LIN {X 0,Y 225.731,Z 1154.757,A -85,B 0,C 180,E1 26958.858,E2 26958.858} C_VEL
LIN {X 0,Y 255.591,Z 1130.454,A -85,B 0,C 180,E1 26969.522,E2 26969.522} C_VEL
LIN {X 0,Y 287.128,Z 1102.716,A -85,B 0,C 180,E1 26976.829,E2 26976.829} C_VEL
LIN {X 0,Y 319.743,Z 1070.349,A -85,B 0,C 180,E1 26982.239,E2 26982.239} C_VEL
LIN {X 0,Y 351.909,Z 1032.611,A -85,B 0,C 180,E1 26986.269,E2 26986.269} C_VEL
LIN {X 0,Y 368.371,Z 1010.613,A -85,B 0,C 180,E1 26987.946,E2 26987.946} C_VEL
LIN {X 0,Y 369.064,Z 1007.37,A -85,B 0,C 180,E1 26989.314,E2 26989.314} C_VEL
LIN {X 0,Y 369.295,Z 1000.148,A -85,B 0,C 180,E1 26995.312,E2 26995.312} C_VEL
LIN {X 0,Y 369.425,Z 998.78,A -85,B 0,C 180,E1 26997.662,E2 26997.662} C_VEL
LIN {X 0,Y 368.67,Z 999.428,A -85,B 0,C 180,E1 27000.006,E2 27000.006} C_VEL
LIN {X 0,Y 365.941,Z 1005.713,A -85,B 0,C 180,E1 27005.933,E2 27005.933} C_VEL
LIN {X 0,Y 364.301,Z 1009.952,A -85,B 0,C 180,E1 27008.244,E2 27008.244} C_VEL
LIN {X 0,Y 336.486,Z 1043.678,A -85,B 0,C 180,E1 27011.534,E2 27011.534} C_VEL
LIN {X 0,Y 304.444,Z 1075.769,A -85,B 0,C 180,E1 27016.292,E2 27016.292} C_VEL
LIN {X 0,Y 273.32,Z 1102.243,A -85,B 0,C 180,E1 27022.45,E2 27022.45} C_VEL
LIN {X 0,Y 242.415,Z 1124.929,A -85,B 0,C 180,E1 27031.225,E2 27031.225} C_VEL
LIN {X 0,Y 228.244,Z 1134.299,A -85,B 0,C 180,E1 27036.811,E2 27036.811} C_VEL
LIN {X 0,Y 217.232,Z 1139.855,A -85,B 0,C 180,E1 27040.027,E2 27040.027} C_VEL
LIN {X 0,Y 206.835,Z 1144.678,A -85,B 0,C 180,E1 27043.615,E2 27043.615} C_VEL
LIN {X 0,Y 192.084,Z 1153.208,A -85,B 0,C 180,E1 27056.588,E2 27056.588} C_VEL
LIN {X 0,Y 184.823,Z 1157.192,A -85,B 0,C 180,E1 27070.913,E2 27070.913} C_VEL
LIN {X 0,Y 183.688,Z 1157.067,A -85,B 0,C 180,E1 27080.911,E2 27080.911} C_VEL
LIN {X 0,Y 184.934,Z 1155.178,A -85,B 0,C 180,E1 27090.002,E2 27090.002} C_VEL
LIN {X 0,Y 189.195,Z 1150.026,A -85,B 0,C 180,E1 27101.521,E2 27101.521} C_VEL
LIN {X 0,Y 199.74,Z 1139.824,A -85,B 0,C 180,E1 27114.27,E2 27114.27} C_VEL
LIN {X 0,Y 218.512,Z 1123.996,A -85,B 0,C 180,E1 27126.005,E2 27126.005} C_VEL
LIN {X 0,Y 244.526,Z 1101.275,A -85,B 0,C 180,E1 27135.925,E2 27135.925} C_VEL
LIN {X 0,Y 271.832,Z 1074.958,A -85,B 0,C 180,E1 27143.048,E2 27143.048} C_VEL
LIN {X 0,Y 300.799,Z 1042.826,A -85,B 0,C 180,E1 27148.655,E2 27148.655} C_VEL
LIN {X 0,Y 327.326,Z 1007.742,A -85,B 0,C 180,E1 27152.712,E2 27152.712} C_VEL
LIN {X 0,Y 337.468,Z 992.575,A -85,B 0,C 180,E1 27154.024,E2 27154.024} C_VEL
LIN {X 0,Y 339.323,Z 979.812,A -85,B 0,C 180,E1 27159.121,E2 27159.121} C_VEL
LIN {X 0,Y 340.418,Z 970.596,A -85,B 0,C 180,E1 27164.546,E2 27164.546} C_VEL
LIN {X 0,Y 341.292,Z 965.531,A -85,B 0,C 180,E1 27169.791,E2 27169.791} C_VEL
LIN {X 0,Y 342.341,Z 964.643,A -85,B 0,C 180,E1 27174.928,E2 27174.928} C_VEL
LIN {X 0,Y 342.913,Z 967.181,A -85,B 0,C 180,E1 27178.73,E2 27178.73} C_VEL
LIN {X 0,Y 343.424,Z 975.954,A -85,B 0,C 180,E1 27184.409,E2 27184.409} C_VEL
LIN {X 0,Y 343.453,Z 988.167,A -85,B 0,C 180,E1 27189.49,E2 27189.49} C_VEL
LIN {X 0,Y 342.79,Z 996.133,A -85,B 0,C 180,E1 27191.913,E2 27191.913} C_VEL
LIN {X 0,Y 317.01,Z 1035.287,A -85,B 0,C 180,E1 27195.203,E2 27195.203} C_VEL
LIN {X 0,Y 288.961,Z 1071.469,A -85,B 0,C 180,E1 27199.722,E2 27199.722} C_VEL
LIN {X 0,Y 259.817,Z 1103.901,A -85,B 0,C 180,E1 27205.948,E2 27205.948} C_VEL
LIN {X 0,Y 232.582,Z 1131.307,A -85,B 0,C 180,E1 27214.063,E2 27214.063} C_VEL
LIN {X 0,Y 208.777,Z 1154.112,A -85,B 0,C 180,E1 27224.97,E2 27224.97} C_VEL
LIN {X 0,Y 193.756,Z 1169.833,A -85,B 0,C 180,E1 27236.909,E2 27236.909} C_VEL
LIN {X 0,Y 186.533,Z 1179.298,A -85,B 0,C 180,E1 27248.16,E2 27248.16} C_VEL
LIN {X 0,Y 183.801,Z 1185.477,A -85,B 0,C 180,E1 27260.533,E2 27260.533} C_VEL
LIN {X 0,Y 184.143,Z 1187.355,A -85,B 0,C 180,E1 27269.998,E2 27269.998} C_VEL
LIN {X 0,Y 183.626,Z 1186.803,A -85,B 0,C 180,E1 27279.471,E2 27279.471} C_VEL
LIN {X 0,Y 187.317,Z 1181.478,A -85,B 0,C 180,E1 27293.786,E2 27293.786} C_VEL
LIN {X 0,Y 199.841,Z 1170.086,A -85,B 0,C 180,E1 27308.594,E2 27308.594} C_VEL
LIN {X 0,Y 220.297,Z 1154.314,A -85,B 0,C 180,E1 27320.475,E2 27320.475} C_VEL
LIN {X 0,Y 250.559,Z 1130.739,A -85,B 0,C 180,E1 27330.922,E2 27330.922} C_VEL
LIN {X 0,Y 282.961,Z 1103.312,A -85,B 0,C 180,E1 27338.19,E2 27338.19} C_VEL
LIN {X 0,Y 316.996,Z 1070.447,A -85,B 0,C 180,E1 27343.605,E2 27343.605} C_VEL
LIN {X 0,Y 348.412,Z 1034.569,A -85,B 0,C 180,E1 27347.387,E2 27347.387} C_VEL
LIN {X 0,Y 363.267,Z 1015.279,A -85,B 0,C 180,E1 27348.857,E2 27348.857} C_VEL
LIN {X 0,Y 364.088,Z 1012.889,A -85,B 0,C 180,E1 27349.809,E2 27349.809} C_VEL
LIN {X 0,Y 364.525,Z 1006.563,A -85,B 0,C 180,E1 27355.251,E2 27355.251} C_VEL
LIN {X 0,Y 364.682,Z 1005.142,A -85,B 0,C 180,E1 27357.632,E2 27357.632} C_VEL
LIN {X 0,Y 362.859,Z 1007.313,A -85,B 0,C 180,E1 27361.884,E2 27361.884} C_VEL
LIN {X 0,Y 360.058,Z 1014.019,A -85,B 0,C 180,E1 27367.24,E2 27367.24} C_VEL
LIN {X 0,Y 330.698,Z 1048.189,A -85,B 0,C 180,E1 27370.659,E2 27370.659} C_VEL
LIN {X 0,Y 297.895,Z 1079.882,A -85,B 0,C 180,E1 27375.467,E2 27375.467} C_VEL
LIN {X 0,Y 266.374,Z 1105.375,A -85,B 0,C 180,E1 27381.653,E2 27381.653} C_VEL
LIN {X 0,Y 236.474,Z 1126.44,A -85,B 0,C 180,E1 27390.032,E2 27390.032} C_VEL
LIN {X 0,Y 210.577,Z 1142.41,A -85,B 0,C 180,E1 27401.326,E2 27401.326} C_VEL
LIN {X 0,Y 206.835,Z 1144.678,A -85,B 0,C 180,E1 27403.615,E2 27403.615} C_VEL
LIN {X 0,Y 197.08,Z 1148.854,A -85,B 0,C 180,E1 27407.583,E2 27407.583} C_VEL
LIN {X 0,Y 188.062,Z 1152.273,A -85,B 0,C 180,E1 27411.94,E2 27411.94} C_VEL
LIN {X 0,Y 178.94,Z 1157.001,A -85,B 0,C 180,E1 27425.026,E2 27425.026} C_VEL
LIN {X 0,Y 176.095,Z 1158.029,A -85,B 0,C 180,E1 27435.084,E2 27435.084} C_VEL
LIN {X 0,Y 176.124,Z 1157.066,A -85,B 0,C 180,E1 27445.08,E2 27445.08} C_VEL
LIN {X 0,Y 179.237,Z 1153.177,A -85,B 0,C 180,E1 27457.268,E2 27457.268} C_VEL
LIN {X 0,Y 188.287,Z 1144.419,A -85,B 0,C 180,E1 27471.174,E2 27471.174} C_VEL
LIN {X 0,Y 205.027,Z 1130.704,A -85,B 0,C 180,E1 27483.56,E2 27483.56} C_VEL
LIN {X 0,Y 231.034,Z 1109.426,A -85,B 0,C 180,E1 27494.681,E2 27494.681} C_VEL
LIN {X 0,Y 259.187,Z 1083.962,A -85,B 0,C 180,E1 27502.599,E2 27502.599} C_VEL
LIN {X 0,Y 287.826,Z 1054.539,A -85,B 0,C 180,E1 27508.413,E2 27508.413} C_VEL
LIN {X 0,Y 317.766,Z 1017.751,A -85,B 0,C 180,E1 27513.119,E2 27513.119} C_VEL
LIN {X 0,Y 332.912,Z 995.879,A -85,B 0,C 180,E1 27515.209,E2 27515.209} C_VEL
LIN {X 0,Y 334.922,Z 984.233,A -85,B 0,C 180,E1 27520.277,E2 27520.277} C_VEL
LIN {X 0,Y 336.156,Z 975.928,A -85,B 0,C 180,E1 27525.678,E2 27525.678} C_VEL
LIN {X 0,Y 337.207,Z 972.067,A -85,B 0,C 180,E1 27530.37,E2 27530.37} C_VEL
LIN {X 0,Y 338.186,Z 971.363,A -85,B 0,C 180,E1 27534.866,E2 27534.866} C_VEL
LIN {X 0,Y 338.706,Z 973.965,A -85,B 0,C 180,E1 27538.715,E2 27538.715} C_VEL
LIN {X 0,Y 338.891,Z 982.852,A -85,B 0,C 180,E1 27544.469,E2 27544.469} C_VEL
LIN {X 0,Y 338.543,Z 995.446,A -85,B 0,C 180,E1 27549.629,E2 27549.629} C_VEL
LIN {X 0,Y 337.882,Z 999.689,A -85,B 0,C 180,E1 27550.903,E2 27550.903} C_VEL
LIN {X 0,Y 309.246,Z 1041.451,A -85,B 0,C 180,E1 27554.497,E2 27554.497} C_VEL
LIN {X 0,Y 279.64,Z 1077.497,A -85,B 0,C 180,E1 27559.272,E2 27559.272} C_VEL
LIN {X 0,Y 251.113,Z 1107.96,A -85,B 0,C 180,E1 27565.486,E2 27565.486} C_VEL
LIN {X 0,Y 222.993,Z 1134.715,A -85,B 0,C 180,E1 27574.064,E2 27574.064} C_VEL
LIN {X 0,Y 199.803,Z 1156.182,A -85,B 0,C 180,E1 27585.154,E2 27585.154} C_VEL
LIN {X 0,Y 183.614,Z 1172.48,A -85,B 0,C 180,E1 27599.322,E2 27599.322} C_VEL
LIN {X 0,Y 177.133,Z 1181.607,A -85,B 0,C 180,E1 27612.625,E2 27612.625} C_VEL
LIN {X 0,Y 175.787,Z 1185.998,A -85,B 0,C 180,E1 27625.066,E2 27625.066} C_VEL
LIN {X 0,Y 176.27,Z 1186.693,A -85,B 0,C 180,E1 27629.998,E2 27629.998} C_VEL
LIN {X 0,Y 175.744,Z 1186.154,A -85,B 0,C 180,E1 27639.9,E2 27639.9} C_VEL
LIN {X 0,Y 179.846,Z 1180.886,A -85,B 0,C 180,E1 27654.839,E2 27654.839} C_VEL
LIN {X 0,Y 193.381,Z 1169.535,A -85,B 0,C 180,E1 27670.138,E2 27670.138} C_VEL
LIN {X 0,Y 216.929,Z 1152.407,A -85,B 0,C 180,E1 27683,E2 27683} C_VEL
LIN {X 0,Y 247.722,Z 1129.486,A -85,B 0,C 180,E1 27692.909,E2 27692.909} C_VEL
LIN {X 0,Y 280.898,Z 1102.184,A -85,B 0,C 180,E1 27699.931,E2 27699.931} C_VEL
LIN {X 0,Y 314.777,Z 1070.205,A -85,B 0,C 180,E1 27705.039,E2 27705.039} C_VEL
LIN {X 0,Y 346.723,Z 1034.468,A -85,B 0,C 180,E1 27708.702,E2 27708.702} C_VEL
LIN {X 0,Y 358.957,Z 1018.778,A -85,B 0,C 180,E1 27710.007,E2 27710.007} C_VEL
LIN {X 0,Y 359.519,Z 1012.804,A -85,B 0,C 180,E1 27715.184,E2 27715.184} C_VEL
LIN {X 0,Y 359.717,Z 1011.351,A -85,B 0,C 180,E1 27717.599,E2 27717.599} C_VEL
LIN {X 0,Y 358.821,Z 1012.013,A -85,B 0,C 180,E1 27720.007,E2 27720.007} C_VEL
LIN {X 0,Y 355.697,Z 1018.071,A -85,B 0,C 180,E1 27725.824,E2 27725.824} C_VEL
LIN {X 0,Y 354.503,Z 1019.844,A -85,B 0,C 180,E1 27726.44,E2 27726.44} C_VEL
LIN {X 0,Y 324.04,Z 1053.622,A -85,B 0,C 180,E1 27729.87,E2 27729.87} C_VEL
LIN {X 0,Y 293.44,Z 1082.113,A -85,B 0,C 180,E1 27734.272,E2 27734.272} C_VEL
LIN {X 0,Y 258.884,Z 1108.955,A -85,B 0,C 180,E1 27740.948,E2 27740.948} C_VEL
LIN {X 0,Y 228.53,Z 1129.114,A -85,B 0,C 180,E1 27749.483,E2 27749.483} C_VEL
LIN {X 0,Y 201.7,Z 1144.875,A -85,B 0,C 180,E1 27761.482,E2 27761.482} C_VEL
LIN {X 0,Y 188.062,Z 1152.273,A -85,B 0,C 180,E1 27771.94,E2 27771.94} C_VEL
LIN {X 0,Y 182.293,Z 1154.397,A -85,B 0,C 180,E1 27775.515,E2 27775.515} C_VEL
LIN {X 0,Y 173.01,Z 1156.924,A -85,B 0,C 180,E1 27781.105,E2 27781.105} C_VEL
LIN {X 0,Y 172.518,Z 1157.109,A -85,B 0,C 180,E1 27781.812,E2 27781.812} C_VEL
LIN {X 0,Y 168.284,Z 1158.679,A -85,B 0,C 180,E1 27794.375,E2 27794.375} C_VEL
LIN {X 0,Y 168.189,Z 1157.771,A -85,B 0,C 180,E1 27804.848,E2 27804.848} C_VEL
LIN {X 0,Y 171.444,Z 1153.939,A -85,B 0,C 180,E1 27817.6,E2 27817.6} C_VEL
LIN {X 0,Y 180.976,Z 1145.25,A -85,B 0,C 180,E1 27832.073,E2 27832.073} C_VEL
LIN {X 0,Y 198.518,Z 1131.649,A -85,B 0,C 180,E1 27844.816,E2 27844.816} C_VEL
LIN {X 0,Y 225.53,Z 1110.45,A -85,B 0,C 180,E1 27856.081,E2 27856.081} C_VEL
LIN {X 0,Y 254.512,Z 1085.139,A -85,B 0,C 180,E1 27863.998,E2 27863.998} C_VEL
LIN {X 0,Y 284.131,Z 1055.549,A -85,B 0,C 180,E1 27869.799,E2 27869.799} C_VEL
LIN {X 0,Y 314.371,Z 1019.202,A -85,B 0,C 180,E1 27874.382,E2 27874.382} C_VEL
LIN {X 0,Y 327.409,Z 1001.32,A -85,B 0,C 180,E1 27876.004,E2 27876.004} C_VEL
LIN {X 0,Y 328.56,Z 998.218,A -85,B 0,C 180,E1 27876.907,E2 27876.907} C_VEL
LIN {X 0,Y 330.956,Z 986.563,A -85,B 0,C 180,E1 27882.729,E2 27882.729} C_VEL
LIN {X 0,Y 332.263,Z 980.103,A -85,B 0,C 180,E1 27888.183,E2 27888.183} C_VEL
LIN {X 0,Y 333.478,Z 978.043,A -85,B 0,C 180,E1 27893.438,E2 27893.438} C_VEL
LIN {X 0,Y 334.375,Z 979.22,A -85,B 0,C 180,E1 27897.403,E2 27897.403} C_VEL
LIN {X 0,Y 334.251,Z 987.229,A -85,B 0,C 180,E1 27903.233,E2 27903.233} C_VEL
LIN {X 0,Y 333.666,Z 998.99,A -85,B 0,C 180,E1 27908.457,E2 27908.457} C_VEL
LIN {X 0,Y 333.359,Z 1002.551,A -85,B 0,C 180,E1 27909.78,E2 27909.78} C_VEL
LIN {X 0,Y 304.76,Z 1043.252,A -85,B 0,C 180,E1 27913.316,E2 27913.316} C_VEL
LIN {X 0,Y 273.281,Z 1080.243,A -85,B 0,C 180,E1 27918.274,E2 27918.274} C_VEL
LIN {X 0,Y 243.35,Z 1110.799,A -85,B 0,C 180,E1 27924.742,E2 27924.742} C_VEL
LIN {X 0,Y 213.562,Z 1137.974,A -85,B 0,C 180,E1 27934.001,E2 27934.001} C_VEL
LIN {X 0,Y 190.625,Z 1158.131,A -85,B 0,C 180,E1 27945.5,E2 27945.5} C_VEL
LIN {X 0,Y 175.419,Z 1172.928,A -85,B 0,C 180,E1 27959.454,E2 27959.454} C_VEL
LIN {X 0,Y 169.44,Z 1180.852,A -85,B 0,C 180,E1 27971.809,E2 27971.809} C_VEL
LIN {X 0,Y 167.885,Z 1185.307,A -85,B 0,C 180,E1 27984.833,E2 27984.833} C_VEL
LIN {X 0,Y 168.375,Z 1186.03,A -85,B 0,C 180,E1 27989.997,E2 27989.997} C_VEL
LIN {X 0,Y 167.888,Z 1185.507,A -85,B 0,C 180,E1 28000.368,E2 28000.368} C_VEL
LIN {X 0,Y 172.441,Z 1180.296,A -85,B 0,C 180,E1 28015.984,E2 28015.984} C_VEL
LIN {X 0,Y 187.013,Z 1169.049,A -85,B 0,C 180,E1 28031.715,E2 28031.715} C_VEL
LIN {X 0,Y 210.887,Z 1152.735,A -85,B 0,C 180,E1 28044.367,E2 28044.367} C_VEL
LIN {X 0,Y 244.692,Z 1128.602,A -85,B 0,C 180,E1 28054.817,E2 28054.817} C_VEL
LIN {X 0,Y 278.629,Z 1101.448,A -85,B 0,C 180,E1 28061.631,E2 28061.631} C_VEL
LIN {X 0,Y 314.428,Z 1068.351,A -85,B 0,C 180,E1 28066.701,E2 28066.701} C_VEL
LIN {X 0,Y 348.48,Z 1030.407,A -85,B 0,C 180,E1 28070.341,E2 28070.341} C_VEL
LIN {X 0,Y 353.938,Z 1023.696,A -85,B 0,C 180,E1 28070.868,E2 28070.868} C_VEL
LIN {X 0,Y 354.461,Z 1019.006,A -85,B 0,C 180,E1 28075.115,E2 28075.115} C_VEL
LIN {X 0,Y 354.688,Z 1017.501,A -85,B 0,C 180,E1 28077.565,E2 28077.565} C_VEL
LIN {X 0,Y 353.016,Z 1019.198,A -85,B 0,C 180,E1 28081.233,E2 28081.233} C_VEL
LIN {X 0,Y 350.663,Z 1023.307,A -85,B 0,C 180,E1 28085.231,E2 28085.231} C_VEL
LIN {X 0,Y 319.094,Z 1057.396,A -85,B 0,C 180,E1 28088.854,E2 28088.854} C_VEL
LIN {X 0,Y 285.521,Z 1087.118,A -85,B 0,C 180,E1 28093.605,E2 28093.605} C_VEL
LIN {X 0,Y 253.013,Z 1111.397,A -85,B 0,C 180,E1 28099.843,E2 28099.843} C_VEL
LIN {X 0,Y 221.711,Z 1131.129,A -85,B 0,C 180,E1 28108.509,E2 28108.509} C_VEL
LIN {X 0,Y 196.209,Z 1145.373,A -85,B 0,C 180,E1 28119.635,E2 28119.635} C_VEL
LIN {X 0,Y 178.328,Z 1154.355,A -85,B 0,C 180,E1 28133.621,E2 28133.621} C_VEL
LIN {X 0,Y 172.518,Z 1157.109,A -85,B 0,C 180,E1 28141.812,E2 28141.812} C_VEL
LIN {X 0,Y 167.988,Z 1158.233,A -85,B 0,C 180,E1 28145.949,E2 28145.949} C_VEL
LIN {X 0,Y 160.783,Z 1159.292,A -85,B 0,C 180,E1 28152.412,E2 28152.412} C_VEL
LIN {X 0,Y 160.57,Z 1159.316,A -85,B 0,C 180,E1 28153.195,E2 28153.195} C_VEL
LIN {X 0,Y 160.265,Z 1158.474,A -85,B 0,C 180,E1 28164.592,E2 28164.592} C_VEL
LIN {X 0,Y 163.674,Z 1154.698,A -85,B 0,C 180,E1 28177.963,E2 28177.963} C_VEL
LIN {X 0,Y 173.716,Z 1146.077,A -85,B 0,C 180,E1 28193.047,E2 28193.047} C_VEL
LIN {X 0,Y 192.116,Z 1132.592,A -85,B 0,C 180,E1 28206.155,E2 28206.155} C_VEL
LIN {X 0,Y 220.164,Z 1111.474,A -85,B 0,C 180,E1 28217.551,E2 28217.551} C_VEL
LIN {X 0,Y 249.998,Z 1086.315,A -85,B 0,C 180,E1 28225.447,E2 28225.447} C_VEL
LIN {X 0,Y 280.296,Z 1056.832,A -85,B 0,C 180,E1 28231.175,E2 28231.175} C_VEL
LIN {X 0,Y 310.571,Z 1021.366,A -85,B 0,C 180,E1 28235.6,E2 28235.6} C_VEL
LIN {X 0,Y 323.505,Z 1003.782,A -85,B 0,C 180,E1 28237.325,E2 28237.325} C_VEL
LIN {X 0,Y 326.234,Z 992.448,A -85,B 0,C 180,E1 28243.148,E2 28243.148} C_VEL
LIN {X 0,Y 327.846,Z 986.527,A -85,B 0,C 180,E1 28248.396,E2 28248.396} C_VEL
LIN {X 0,Y 329.032,Z 984.615,A -85,B 0,C 180,E1 28253.473,E2 28253.473} C_VEL
LIN {X 0,Y 329.875,Z 985.796,A -85,B 0,C 180,E1 28257.367,E2 28257.367} C_VEL
LIN {X 0,Y 329.614,Z 994.014,A -85,B 0,C 180,E1 28263.278,E2 28263.278} C_VEL
LIN {X 0,Y 328.439,Z 1006.01,A -85,B 0,C 180,E1 28268.593,E2 28268.593} C_VEL
LIN {X 0,Y 322.913,Z 1014.638,A -85,B 0,C 180,E1 28269.365,E2 28269.365} C_VEL
LIN {X 0,Y 293.321,Z 1053.597,A -85,B 0,C 180,E1 28273.105,E2 28273.105} C_VEL
LIN {X 0,Y 263.005,Z 1087.06,A -85,B 0,C 180,E1 28277.975,E2 28277.975} C_VEL
LIN {X 0,Y 230.898,Z 1117.905,A -85,B 0,C 180,E1 28285.168,E2 28285.168} C_VEL
LIN {X 0,Y 202.269,Z 1142.521,A -85,B 0,C 180,E1 28294.731,E2 28294.731} C_VEL
LIN {X 0,Y 179.093,Z 1162.144,A -85,B 0,C 180,E1 28307.542,E2 28307.542} C_VEL
LIN {X 0,Y 165.168,Z 1175.494,A -85,B 0,C 180,E1 28322.774,E2 28322.774} C_VEL
LIN {X 0,Y 161.072,Z 1181.398,A -85,B 0,C 180,E1 28333.65,E2 28333.65} C_VEL
LIN {X 0,Y 160.001,Z 1184.616,A -85,B 0,C 180,E1 28344.578,E2 28344.578} C_VEL
LIN {X 0,Y 160.497,Z 1185.368,A -85,B 0,C 180,E1 28349.997,E2 28349.997} C_VEL
LIN {X 0,Y 160.014,Z 1184.857,A -85,B 0,C 180,E1 28360.884,E2 28360.884} C_VEL
LIN {X 0,Y 163.659,Z 1180.889,A -85,B 0,C 180,E1 28374.548,E2 28374.548} C_VEL
LIN {X 0,Y 177.039,Z 1171.082,A -85,B 0,C 180,E1 28390.629,E2 28390.629} C_VEL
LIN {X 0,Y 202.91,Z 1154.305,A -85,B 0,C 180,E1 28405.001,E2 28405.001} C_VEL
LIN {X 0,Y 233.771,Z 1133.521,A -85,B 0,C 180,E1 28414.816,E2 28414.816} C_VEL
LIN {X 0,Y 271.366,Z 1105.178,A -85,B 0,C 180,E1 28422.476,E2 28422.476} C_VEL
LIN {X 0,Y 306.396,Z 1074.104,A -85,B 0,C 180,E1 28427.433,E2 28427.433} C_VEL
LIN {X 0,Y 339.612,Z 1039.409,A -85,B 0,C 180,E1 28430.956,E2 28430.956} C_VEL
LIN {X 0,Y 348.77,Z 1028.328,A -85,B 0,C 180,E1 28431.912,E2 28431.912} C_VEL
LIN {X 0,Y 349.574,Z 1023.585,A -85,B 0,C 180,E1 28437.529,E2 28437.529} C_VEL
LIN {X 0,Y 347.647,Z 1025.284,A -85,B 0,C 180,E1 28441.345,E2 28441.345} C_VEL
LIN {X 0,Y 345.198,Z 1028.984,A -85,B 0,C 180,E1 28444.489,E2 28444.489} C_VEL
LIN {X 0,Y 313.827,Z 1061.414,A -85,B 0,C 180,E1 28447.869,E2 28447.869} C_VEL
LIN {X 0,Y 277.21,Z 1092.485,A -85,B 0,C 180,E1 28452.999,E2 28452.999} C_VEL
LIN {X 0,Y 244.236,Z 1115.586,A -85,B 0,C 180,E1 28459.35,E2 28459.35} C_VEL
LIN {X 0,Y 212.851,Z 1134.372,A -85,B 0,C 180,E1 28468.211,E2 28468.211} C_VEL
LIN {X 0,Y 185.812,Z 1148.264,A -85,B 0,C 180,E1 28480.605,E2 28480.605} C_VEL
LIN {X 0,Y 170.981,Z 1155.239,A -85,B 0,C 180,E1 28492.72,E2 28492.72} C_VEL
LIN {X 0,Y 161.887,Z 1159.059,A -85,B 0,C 180,E1 28508.079,E2 28508.079} C_VEL
LIN {X 0,Y 160.57,Z 1159.316,A -85,B 0,C 180,E1 28513.195,E2 28513.195} C_VEL
LIN {X 0,Y 157.62,Z 1159.481,A -85,B 0,C 180,E1 28517.785,E2 28517.785} C_VEL
LIN {X 0,Y 152.427,Z 1158.913,A -85,B 0,C 180,E1 28525.724,E2 28525.724} C_VEL
LIN {X 0,Y 155.909,Z 1155.455,A -85,B 0,C 180,E1 28538.362,E2 28538.362} C_VEL
LIN {X 0,Y 166.498,Z 1146.905,A -85,B 0,C 180,E1 28554.108,E2 28554.108} C_VEL
LIN {X 0,Y 185.828,Z 1133.532,A -85,B 0,C 180,E1 28567.584,E2 28567.584} C_VEL
LIN {X 0,Y 214.946,Z 1112.5,A -85,B 0,C 180,E1 28579.094,E2 28579.094} C_VEL
LIN {X 0,Y 244.258,Z 1088.734,A -85,B 0,C 180,E1 28586.639,E2 28586.639} C_VEL
LIN {X 0,Y 276.622,Z 1058.104,A -85,B 0,C 180,E1 28592.589,E2 28592.589} C_VEL
LIN {X 0,Y 307.077,Z 1023.329,A -85,B 0,C 180,E1 28596.867,E2 28596.867} C_VEL
LIN {X 0,Y 318.503,Z 1008.421,A -85,B 0,C 180,E1 28598.213,E2 28598.213} C_VEL
LIN {X 0,Y 321.24,Z 999.294,A -85,B 0,C 180,E1 28602.944,E2 28602.944} C_VEL
LIN {X 0,Y 323.363,Z 992.625,A -85,B 0,C 180,E1 28608.928,E2 28608.928} C_VEL
LIN {X 0,Y 324.977,Z 991.085,A -85,B 0,C 180,E1 28614.656,E2 28614.656} C_VEL
LIN {X 0,Y 325.234,Z 993.789,A -85,B 0,C 180,E1 28618.661,E2 28618.661} C_VEL
LIN {X 0,Y 324.548,Z 1001.888,A -85,B 0,C 180,E1 28623.998,E2 28623.998} C_VEL
LIN {X 0,Y 323.598,Z 1009.894,A -85,B 0,C 180,E1 28627.53,E2 28627.53} C_VEL
LIN {X 0,Y 305.45,Z 1034.936,A -85,B 0,C 180,E1 28629.717,E2 28629.717} C_VEL
LIN {X 0,Y 275.803,Z 1070.013,A -85,B 0,C 180,E1 28633.717,E2 28633.717} C_VEL
LIN {X 0,Y 243.179,Z 1102.545,A -85,B 0,C 180,E1 28639.579,E2 28639.579} C_VEL
LIN {X 0,Y 212.136,Z 1129.746,A -85,B 0,C 180,E1 28647.568,E2 28647.568} C_VEL
LIN {X 0,Y 184.072,Z 1152.251,A -85,B 0,C 180,E1 28658.86,E2 28658.86} C_VEL
LIN {X 0,Y 164.209,Z 1168.685,A -85,B 0,C 180,E1 28673.259,E2 28673.259} C_VEL
LIN {X 0,Y 155.134,Z 1177.976,A -85,B 0,C 180,E1 28687.065,E2 28687.065} C_VEL
LIN {X 0,Y 152.343,Z 1182.585,A -85,B 0,C 180,E1 28698.555,E2 28698.555} C_VEL
LIN {X 0,Y 152.598,Z 1184.704,A -85,B 0,C 180,E1 28709.997,E2 28709.997} C_VEL
LIN {X 0,Y 152.152,Z 1184.207,A -85,B 0,C 180,E1 28721.454,E2 28721.454} C_VEL
LIN {X 0,Y 157.847,Z 1179.117,A -85,B 0,C 180,E1 28738.595,E2 28738.595} C_VEL
LIN {X 0,Y 175.559,Z 1167.585,A -85,B 0,C 180,E1 28755.756,E2 28755.756} C_VEL
LIN {X 0,Y 202.041,Z 1151.475,A -85,B 0,C 180,E1 28768.442,E2 28768.442} C_VEL
LIN {X 0,Y 239.244,Z 1126.966,A -85,B 0,C 180,E1 28778.747,E2 28778.747} C_VEL
LIN {X 0,Y 275.474,Z 1099.471,A -85,B 0,C 180,E1 28785.195,E2 28785.195} C_VEL
LIN {X 0,Y 311.942,Z 1067.088,A -85,B 0,C 180,E1 28789.74,E2 28789.74} C_VEL
LIN {X 0,Y 342.597,Z 1034.372,A -85,B 0,C 180,E1 28792.701,E2 28792.701} C_VEL
LIN {X 0,Y 343.582,Z 1032.961,A -85,B 0,C 180,E1 28793.06,E2 28793.06} C_VEL
LIN {X 0,Y 344.281,Z 1029.495,A -85,B 0,C 180,E1 28797.491,E2 28797.491} C_VEL
LIN {X 0,Y 342.29,Z 1031.261,A -85,B 0,C 180,E1 28801.366,E2 28801.366} C_VEL
LIN {X 0,Y 341.056,Z 1033.101,A -85,B 0,C 180,E1 28803.316,E2 28803.316} C_VEL
LIN {X 0,Y 306.4,Z 1067.333,A -85,B 0,C 180,E1 28807.105,E2 28807.105} C_VEL
LIN {X 0,Y 272.095,Z 1095.226,A -85,B 0,C 180,E1 28811.817,E2 28811.817} C_VEL
LIN {X 0,Y 236.12,Z 1119.324,A -85,B 0,C 180,E1 28818.674,E2 28818.674} C_VEL
LIN {X 0,Y 204.662,Z 1137.028,A -85,B 0,C 180,E1 28827.627,E2 28827.627} C_VEL
LIN {X 0,Y 177.843,Z 1149.973,A -85,B 0,C 180,E1 28840.121,E2 28840.121} C_VEL
LIN {X 0,Y 160.446,Z 1157.455,A -85,B 0,C 180,E1 28855.594,E2 28855.594} C_VEL
LIN {X 0,Y 154.33,Z 1159.682,A -85,B 0,C 180,E1 28866.945,E2 28866.945} C_VEL
LIN {X 0,Y 152.211,Z 1159.383,A -85,B 0,C 180,E1 28883.256,E2 28883.256} C_VEL
LIN {X 0,Y 152.427,Z 1158.913,A -85,B 0,C 180,E1 28885.724,E2 28885.724} C_VEL
LIN {X 0,Y 150.864,Z 1158.162,A -85,B 0,C 180,E1 28890.625,E2 28890.625} C_VEL
LIN {X 0,Y 148.228,Z 1156.14,A -85,B 0,C 180,E1 28898.991,E2 28898.991} C_VEL
LIN {X 0,Y 158.966,Z 1148.005,A -85,B 0,C 180,E1 28914.869,E2 28914.869} C_VEL
LIN {X 0,Y 179.659,Z 1134.448,A -85,B 0,C 180,E1 28929.115,E2 28929.115} C_VEL
LIN {X 0,Y 207.328,Z 1115.366,A -85,B 0,C 180,E1 28939.937,E2 28939.937} C_VEL
LIN {X 0,Y 238.602,Z 1091.155,A -85,B 0,C 180,E1 28947.898,E2 28947.898} C_VEL
LIN {X 0,Y 271.57,Z 1060.9,A -85,B 0,C 180,E1 28953.804,E2 28953.804} C_VEL
LIN {X 0,Y 301.338,Z 1028.256,A -85,B 0,C 180,E1 28957.884,E2 28957.884} C_VEL
LIN {X 0,Y 313.435,Z 1013.06,A -85,B 0,C 180,E1 28959.266,E2 28959.266} C_VEL
LIN {X 0,Y 315.581,Z 1007.495,A -85,B 0,C 180,E1 28961.868,E2 28961.868} C_VEL
LIN {X 0,Y 317.601,Z 1001.486,A -85,B 0,C 180,E1 28966.229,E2 28966.229} C_VEL
LIN {X 0,Y 319.447,Z 997.685,A -85,B 0,C 180,E1 28971.834,E2 28971.834} C_VEL
LIN {X 0,Y 320.246,Z 997.416,A -85,B 0,C 180,E1 28974.577,E2 28974.577} C_VEL
LIN {X 0,Y 320.428,Z 1000.169,A -85,B 0,C 180,E1 28978.641,E2 28978.641} C_VEL
LIN {X 0,Y 319.516,Z 1008.587,A -85,B 0,C 180,E1 28984.061,E2 28984.061} C_VEL
LIN {X 0,Y 318.731,Z 1013.6,A -85,B 0,C 180,E1 28986.384,E2 28986.384} C_VEL
LIN {X 0,Y 313.304,Z 1021.394,A -85,B 0,C 180,E1 28987.139,E2 28987.139} C_VEL
LIN {X 0,Y 283.953,Z 1057.661,A -85,B 0,C 180,E1 28990.633,E2 28990.633} C_VEL
LIN {X 0,Y 249.498,Z 1093.063,A -85,B 0,C 180,E1 28995.945,E2 28995.945} C_VEL
LIN {X 0,Y 218.198,Z 1120.642,A -85,B 0,C 180,E1 29002.765,E2 29002.765} C_VEL
LIN {X 0,Y 188.236,Z 1144.307,A -85,B 0,C 180,E1 29012.546,E2 29012.546} C_VEL
LIN {X 0,Y 163.666,Z 1162.937,A -85,B 0,C 180,E1 29026.17,E2 29026.17} C_VEL
LIN {X 0,Y 149.055,Z 1175.642,A -85,B 0,C 180,E1 29042.854,E2 29042.854} C_VEL
LIN {X 0,Y 144.493,Z 1181.859,A -85,B 0,C 180,E1 29057.924,E2 29057.924} C_VEL
LIN {X 0,Y 144.698,Z 1184.04,A -85,B 0,C 180,E1 29069.997,E2 29069.997} C_VEL
LIN {X 0,Y 144.297,Z 1183.557,A -85,B 0,C 180,E1 29082.087,E2 29082.087} C_VEL
LIN {X 0,Y 148.939,Z 1179.664,A -85,B 0,C 180,E1 29097.163,E2 29097.163} C_VEL
LIN {X 0,Y 163.886,Z 1170.538,A -85,B 0,C 180,E1 29113.745,E2 29113.745} C_VEL
LIN {X 0,Y 191.269,Z 1154.76,A -85,B 0,C 180,E1 29128.132,E2 29128.132} C_VEL
LIN {X 0,Y 225.669,Z 1133.736,A -85,B 0,C 180,E1 29138.29,E2 29138.29} C_VEL
LIN {X 0,Y 265.162,Z 1105.752,A -85,B 0,C 180,E1 29145.646,E2 29145.646} C_VEL
LIN {X 0,Y 300.139,Z 1076.554,A -85,B 0,C 180,E1 29150.131,E2 29150.131} C_VEL
LIN {X 0,Y 337.225,Z 1039.352,A -85,B 0,C 180,E1 29153.674,E2 29153.674} C_VEL
LIN {X 0,Y 338.412,Z 1037.756,A -85,B 0,C 180,E1 29154.21,E2 29154.21} C_VEL
LIN {X 0,Y 338.974,Z 1035.421,A -85,B 0,C 180,E1 29157.452,E2 29157.452} C_VEL
LIN {X 0,Y 336.415,Z 1037.604,A -85,B 0,C 180,E1 29161.938,E2 29161.938} C_VEL
LIN {X 0,Y 336.205,Z 1037.867,A -85,B 0,C 180,E1 29162.261,E2 29162.261} C_VEL
LIN {X 0,Y 327.312,Z 1047.149,A -85,B 0,C 180,E1 29163.286,E2 29163.286} C_VEL
LIN {X 0,Y 293.067,Z 1078.043,A -85,B 0,C 180,E1 29166.996,E2 29166.996} C_VEL
LIN {X 0,Y 256.34,Z 1105.361,A -85,B 0,C 180,E1 29172.312,E2 29172.312} C_VEL
LIN {X 0,Y 218.83,Z 1128.1,A -85,B 0,C 180,E1 29180.211,E2 29180.211} C_VEL
LIN {X 0,Y 187.465,Z 1143.879,A -85,B 0,C 180,E1 29190.539,E2 29190.539} C_VEL
LIN {X 0,Y 161.509,Z 1155.092,A -85,B 0,C 180,E1 29205.733,E2 29205.733} C_VEL
LIN {X 0,Y 149.668,Z 1159.507,A -85,B 0,C 180,E1 29219.683,E2 29219.683} C_VEL
LIN {X 0,Y 145.062,Z 1160.625,A -85,B 0,C 180,E1 29231.792,E2 29231.792} C_VEL
LIN {X 0,Y 144.551,Z 1159.55,A -85,B 0,C 180,E1 29245.873,E2 29245.873} C_VEL
LIN {X 0,Y 148.228,Z 1156.14,A -85,B 0,C 180,E1 29258.991,E2 29258.991} C_VEL
LIN {X 0,Y 147.483,Z 1153.983,A -85,B 0,C 180,E1 29265.736,E2 29265.736} C_VEL
LIN {X 0,Y 148.452,Z 1151.102,A -85,B 0,C 180,E1 29272.47,E2 29272.47} C_VEL
LIN {X 0,Y 167.527,Z 1139.098,A -85,B 0,C 180,E1 29287.511,E2 29287.511} C_VEL
LIN {X 0,Y 197.205,Z 1120.057,A -85,B 0,C 180,E1 29300.024,E2 29300.024} C_VEL
LIN {X 0,Y 231.587,Z 1094.595,A -85,B 0,C 180,E1 29308.92,E2 29308.92} C_VEL
LIN {X 0,Y 262.711,Z 1067.497,A -85,B 0,C 180,E1 29314.491,E2 29314.491} C_VEL
LIN {X 0,Y 296.787,Z 1031.815,A -85,B 0,C 180,E1 29319.053,E2 29319.053} C_VEL
LIN {X 0,Y 309.142,Z 1016.821,A -85,B 0,C 180,E1 29320.42,E2 29320.42} C_VEL
LIN {X 0,Y 311.81,Z 1009.792,A -85,B 0,C 180,E1 29324.534,E2 29324.534} C_VEL
LIN {X 0,Y 313.767,Z 1005.463,A -85,B 0,C 180,E1 29328.885,E2 29328.885} C_VEL
LIN {X 0,Y 315.481,Z 1003.762,A -85,B 0,C 180,E1 29334.495,E2 29334.495} C_VEL
LIN {X 0,Y 315.608,Z 1006.565,A -85,B 0,C 180,E1 29338.621,E2 29338.621} C_VEL
LIN {X 0,Y 314.495,Z 1013.786,A -85,B 0,C 180,E1 29343.436,E2 29343.436} C_VEL
LIN {X 0,Y 313.179,Z 1018.664,A -85,B 0,C 180,E1 29345.53,E2 29345.53} C_VEL
LIN {X 0,Y 282.792,Z 1055.993,A -85,B 0,C 180,E1 29348.911,E2 29348.911} C_VEL
LIN {X 0,Y 248.934,Z 1090.242,A -85,B 0,C 180,E1 29353.762,E2 29353.762} C_VEL
LIN {X 0,Y 215.843,Z 1118.921,A -85,B 0,C 180,E1 29360.479,E2 29360.479} C_VEL
LIN {X 0,Y 183.163,Z 1143.801,A -85,B 0,C 180,E1 29370.58,E2 29370.58} C_VEL
LIN {X 0,Y 157.73,Z 1162.054,A -85,B 0,C 180,E1 29384.062,E2 29384.062} C_VEL
LIN {X 0,Y 141.816,Z 1174.843,A -85,B 0,C 180,E1 29401.344,E2 29401.344} C_VEL
LIN {X 0,Y 136.668,Z 1181.132,A -85,B 0,C 180,E1 29417.221,E2 29417.221} C_VEL
LIN {X 0,Y 136.796,Z 1183.375,A -85,B 0,C 180,E1 29429.997,E2 29429.997} C_VEL
LIN {X 0,Y 136.467,Z 1182.907,A -85,B 0,C 180,E1 29442.792,E2 29442.792} C_VEL
LIN {X 0,Y 143.626,Z 1177.94,A -85,B 0,C 180,E1 29461.736,E2 29461.736} C_VEL
LIN {X 0,Y 164.498,Z 1166.431,A -85,B 0,C 180,E1 29479.999,E2 29479.999} C_VEL
LIN {X 0,Y 195.166,Z 1149.728,A -85,B 0,C 180,E1 29493.122,E2 29493.122} C_VEL
LIN {X 0,Y 235.249,Z 1125.203,A -85,B 0,C 180,E1 29502.837,E2 29502.837} C_VEL
LIN {X 0,Y 272.942,Z 1097.917,A -85,B 0,C 180,E1 29508.734,E2 29508.734} C_VEL
LIN {X 0,Y 311.427,Z 1064.794,A -85,B 0,C 180,E1 29512.916,E2 29512.916} C_VEL
LIN {X 0,Y 332.974,Z 1042.888,A -85,B 0,C 180,E1 29514.799,E2 29514.799} C_VEL
LIN {X 0,Y 333.444,Z 1041.143,A -85,B 0,C 180,E1 29517.41,E2 29517.41} C_VEL
LIN {X 0,Y 331.225,Z 1042.828,A -85,B 0,C 180,E1 29521.314,E2 29521.314} C_VEL
LIN {X 0,Y 296.917,Z 1074.459,A -85,B 0,C 180,E1 29524.824,E2 29524.824} C_VEL
LIN {X 0,Y 257.9,Z 1103.508,A -85,B 0,C 180,E1 29529.966,E2 29529.966} C_VEL
LIN {X 0,Y 221.092,Z 1125.742,A -85,B 0,C 180,E1 29536.894,E2 29536.894} C_VEL
LIN {X 0,Y 186.526,Z 1143.008,A -85,B 0,C 180,E1 29546.986,E2 29546.986} C_VEL
LIN {X 0,Y 157.189,Z 1154.985,A -85,B 0,C 180,E1 29562.316,E2 29562.316} C_VEL
LIN {X 0,Y 142.56,Z 1160.115,A -85,B 0,C 180,E1 29578.028,E2 29578.028} C_VEL
LIN {X 0,Y 137.361,Z 1161.279,A -85,B 0,C 180,E1 29590.733,E2 29590.733} C_VEL
LIN {X 0,Y 136.586,Z 1160.372,A -85,B 0,C 180,E1 29604.905,E2 29604.905} C_VEL
LIN {X 0,Y 140.474,Z 1156.903,A -85,B 0,C 180,E1 29619.482,E2 29619.482} C_VEL
LIN {X 0,Y 148.452,Z 1151.102,A -85,B 0,C 180,E1 29632.47,E2 29632.47} C_VEL
LIN {X 0,Y 150.551,Z 1148.611,A -85,B 0,C 180,E1 29637.349,E2 29637.349} C_VEL
LIN {X 0,Y 153.788,Z 1144.423,A -85,B 0,C 180,E1 29644.552,E2 29644.552} C_VEL
LIN {X 0,Y 154.758,Z 1143.831,A -85,B 0,C 180,E1 29645.252,E2 29645.252} C_VEL
LIN {X 0,Y 181.98,Z 1127.588,A -85,B 0,C 180,E1 29658.364,E2 29658.364} C_VEL
LIN {X 0,Y 216.582,Z 1104.124,A -85,B 0,C 180,E1 29668.252,E2 29668.252} C_VEL
LIN {X 0,Y 250.708,Z 1076.589,A -85,B 0,C 180,E1 29674.708,E2 29674.708} C_VEL
LIN {X 0,Y 282.986,Z 1045.534,A -85,B 0,C 180,E1 29679.15,E2 29679.15} C_VEL
LIN {X 0,Y 304.615,Z 1020.738,A -85,B 0,C 180,E1 29681.58,E2 29681.58} C_VEL
LIN {X 0,Y 307.265,Z 1014.567,A -85,B 0,C 180,E1 29685.757,E2 29685.757} C_VEL
LIN {X 0,Y 308.607,Z 1011.813,A -85,B 0,C 180,E1 29688.697,E2 29688.697} C_VEL
LIN {X 0,Y 310.57,Z 1010.003,A -85,B 0,C 180,E1 29694.408,E2 29694.408} C_VEL
LIN {X 0,Y 310.575,Z 1012.809,A -85,B 0,C 180,E1 29698.598,E2 29698.598} C_VEL
LIN {X 0,Y 309.06,Z 1020.796,A -85,B 0,C 180,E1 29703.787,E2 29703.787} C_VEL
LIN {X 0,Y 308.883,Z 1021.694,A -85,B 0,C 180,E1 29704.243,E2 29704.243} C_VEL
LIN {X 0,Y 278.125,Z 1058.27,A -85,B 0,C 180,E1 29707.62,E2 29707.62} C_VEL
LIN {X 0,Y 242.613,Z 1093.153,A -85,B 0,C 180,E1 29712.597,E2 29712.597} C_VEL
LIN {X 0,Y 206.831,Z 1122.573,A -85,B 0,C 180,E1 29719.831,E2 29719.831} C_VEL
LIN {X 0,Y 174.519,Z 1145.919,A -85,B 0,C 180,E1 29730.012,E2 29730.012} C_VEL
LIN {X 0,Y 148.336,Z 1163.713,A -85,B 0,C 180,E1 29744.508,E2 29744.508} C_VEL
LIN {X 0,Y 134.65,Z 1174.039,A -85,B 0,C 180,E1 29759.664,E2 29759.664} C_VEL
LIN {X 0,Y 128.847,Z 1180.404,A -85,B 0,C 180,E1 29776.431,E2 29776.431} C_VEL
LIN {X 0,Y 128.915,Z 1182.713,A -85,B 0,C 180,E1 29789.997,E2 29789.997} C_VEL
LIN {X 0,Y 128.641,Z 1182.256,A -85,B 0,C 180,E1 29803.584,E2 29803.584} C_VEL
LIN {X 0,Y 134.571,Z 1178.441,A -85,B 0,C 180,E1 29820.348,E2 29820.348} C_VEL
LIN {X 0,Y 154.275,Z 1168.399,A -85,B 0,C 180,E1 29839.382,E2 29839.382} C_VEL
LIN {X 0,Y 188.454,Z 1150.909,A -85,B 0,C 180,E1 29854.429,E2 29854.429} C_VEL
LIN {X 0,Y 226.399,Z 1128.874,A -85,B 0,C 180,E1 29863.627,E2 29863.627} C_VEL
LIN {X 0,Y 266.177,Z 1101.732,A -85,B 0,C 180,E1 29869.803,E2 29869.803} C_VEL
LIN {X 0,Y 305.625,Z 1069.027,A -85,B 0,C 180,E1 29873.991,E2 29873.991} C_VEL
LIN {X 0,Y 327.229,Z 1048.155,A -85,B 0,C 180,E1 29875.795,E2 29875.795} C_VEL
LIN {X 0,Y 327.857,Z 1046.842,A -85,B 0,C 180,E1 29877.365,E2 29877.365} C_VEL
LIN {X 0,Y 326.311,Z 1047.828,A -85,B 0,C 180,E1 29880.339,E2 29880.339} C_VEL
LIN {X 0,Y 289.317,Z 1080.211,A -85,B 0,C 180,E1 29883.97,E2 29883.97} C_VEL
LIN {X 0,Y 251.774,Z 1106.947,A -85,B 0,C 180,E1 29888.819,E2 29888.819} C_VEL
LIN {X 0,Y 211.661,Z 1129.893,A -85,B 0,C 180,E1 29896.376,E2 29896.376} C_VEL
LIN {X 0,Y 177.456,Z 1145.656,A -85,B 0,C 180,E1 29906.609,E2 29906.609} C_VEL
LIN {X 0,Y 151.179,Z 1155.705,A -85,B 0,C 180,E1 29920.283,E2 29920.283} C_VEL
LIN {X 0,Y 135.604,Z 1160.711,A -85,B 0,C 180,E1 29936.143,E2 29936.143} C_VEL
LIN {X 0,Y 129.721,Z 1161.932,A -85,B 0,C 180,E1 29949.549,E2 29949.549} C_VEL
LIN {X 0,Y 128.552,Z 1161.293,A -85,B 0,C 180,E1 29963.253,E2 29963.253} C_VEL
LIN {X 0,Y 132.671,Z 1157.732,A -85,B 0,C 180,E1 29979.841,E2 29979.841} C_VEL
LIN {X 0,Y 144.258,Z 1150.031,A -85,B 0,C 180,E1 29996.919,E2 29996.919} C_VEL
LIN {X 0,Y 154.758,Z 1143.831,A -85,B 0,C 180,E1 30005.252,E2 30005.252} C_VEL
LIN {X 0,Y 160.246,Z 1139.439,A -85,B 0,C 180,E1 30011.098,E2 30011.098} C_VEL
LIN {X 0,Y 166.913,Z 1134.332,A -85,B 0,C 180,E1 30016.507,E2 30016.507} C_VEL
LIN {X 0,Y 201.546,Z 1112.884,A -85,B 0,C 180,E1 30027.514,E2 30027.514} C_VEL
LIN {X 0,Y 237.949,Z 1085.805,A -85,B 0,C 180,E1 30034.823,E2 30034.823} C_VEL
LIN {X 0,Y 270.351,Z 1056.908,A -85,B 0,C 180,E1 30039.434,E2 30039.434} C_VEL
LIN {X 0,Y 299.026,Z 1026.019,A -85,B 0,C 180,E1 30042.66,E2 30042.66} C_VEL
LIN {X 0,Y 300.477,Z 1023.869,A -85,B 0,C 180,E1 30043.404,E2 30043.404} C_VEL
LIN {X 0,Y 303.427,Z 1018.192,A -85,B 0,C 180,E1 30048.501,E2 30048.501} C_VEL
LIN {X 0,Y 305.516,Z 1016.139,A -85,B 0,C 180,E1 30054.315,E2 30054.315} C_VEL
LIN {X 0,Y 305.551,Z 1018.55,A -85,B 0,C 180,E1 30058.196,E2 30058.196} C_VEL
LIN {X 0,Y 303.987,Z 1025.758,A -85,B 0,C 180,E1 30063.068,E2 30063.068} C_VEL
LIN {X 0,Y 270.944,Z 1063.302,A -85,B 0,C 180,E1 30066.586,E2 30066.586} C_VEL
LIN {X 0,Y 237.232,Z 1095.069,A -85,B 0,C 180,E1 30071.207,E2 30071.207} C_VEL
LIN {X 0,Y 199.445,Z 1125,A -85,B 0,C 180,E1 30078.716,E2 30078.716} C_VEL
LIN {X 0,Y 167.372,Z 1146.908,A -85,B 0,C 180,E1 30088.763,E2 30088.763} C_VEL
LIN {X 0,Y 140.058,Z 1164.554,A -85,B 0,C 180,E1 30104.056,E2 30104.056} C_VEL
LIN {X 0,Y 125.641,Z 1174.901,A -85,B 0,C 180,E1 30121.239,E2 30121.239} C_VEL
LIN {X 0,Y 121.071,Z 1179.677,A -85,B 0,C 180,E1 30135.541,E2 30135.541} C_VEL
LIN {X 0,Y 120.863,Z 1182.066,A -85,B 0,C 180,E1 30150.801,E2 30150.801} C_VEL
LIN {X 0,Y 120.836,Z 1181.605,A -85,B 0,C 180,E1 30164.48,E2 30164.48} C_VEL
LIN {X 0,Y 129.922,Z 1176.759,A -85,B 0,C 180,E1 30185.556,E2 30185.556} C_VEL
LIN {X 0,Y 151.525,Z 1166.642,A -85,B 0,C 180,E1 30203.266,E2 30203.266} C_VEL
LIN {X 0,Y 185.01,Z 1150.425,A -85,B 0,C 180,E1 30216.757,E2 30216.757} C_VEL
LIN {X 0,Y 222.316,Z 1129.639,A -85,B 0,C 180,E1 30225.336,E2 30225.336} C_VEL
LIN {X 0,Y 264.313,Z 1101.813,A -85,B 0,C 180,E1 30231.501,E2 30231.501} C_VEL
LIN {X 0,Y 304.561,Z 1069.111,A -85,B 0,C 180,E1 30235.493,E2 30235.493} C_VEL
LIN {X 0,Y 322.099,Z 1052.634,A -85,B 0,C 180,E1 30236.982,E2 30236.982} C_VEL
LIN {X 0,Y 321.143,Z 1052.873,A -85,B 0,C 180,E1 30239.331,E2 30239.331} C_VEL
LIN {X 0,Y 281.659,Z 1086.046,A -85,B 0,C 180,E1 30243.084,E2 30243.084} C_VEL
LIN {X 0,Y 242.338,Z 1112.271,A -85,B 0,C 180,E1 30248.14,E2 30248.14} C_VEL
LIN {X 0,Y 207.95,Z 1131.058,A -85,B 0,C 180,E1 30254.478,E2 30254.478} C_VEL
LIN {X 0,Y 171.079,Z 1147.218,A -85,B 0,C 180,E1 30265.132,E2 30265.132} C_VEL
LIN {X 0,Y 144.051,Z 1156.894,A -85,B 0,C 180,E1 30279.029,E2 30279.029} C_VEL
LIN {X 0,Y 127.442,Z 1161.654,A -85,B 0,C 180,E1 30296.136,E2 30296.136} C_VEL
LIN {X 0,Y 120.715,Z 1162.523,A -85,B 0,C 180,E1 30315.505,E2 30315.505} C_VEL
LIN {X 0,Y 121.607,Z 1160.914,A -85,B 0,C 180,E1 30330.004,E2 30330.004} C_VEL
LIN {X 0,Y 128.242,Z 1156.227,A -85,B 0,C 180,E1 30347.136,E2 30347.136} C_VEL
LIN {X 0,Y 145.234,Z 1146.453,A -85,B 0,C 180,E1 30364.912,E2 30364.912} C_VEL
LIN {X 0,Y 166.913,Z 1134.332,A -85,B 0,C 180,E1 30376.507,E2 30376.507} C_VEL
LIN {X 0,Y 174.789,Z 1128.783,A -85,B 0,C 180,E1 30381.419,E2 30381.419} C_VEL
LIN {X 0,Y 183.601,Z 1122.602,A -85,B 0,C 180,E1 30385.864,E2 30385.864} C_VEL
LIN {X 0,Y 218.826,Z 1099.056,A -85,B 0,C 180,E1 30393.866,E2 30393.866} C_VEL
LIN {X 0,Y 253.324,Z 1071.496,A -85,B 0,C 180,E1 30399.231,E2 30399.231} C_VEL
LIN {X 0,Y 288.614,Z 1036.721,A -85,B 0,C 180,E1 30403.295,E2 30403.295} C_VEL
LIN {X 0,Y 295.037,Z 1029.554,A -85,B 0,C 180,E1 30403.926,E2 30403.926} C_VEL
LIN {X 0,Y 298.011,Z 1024.432,A -85,B 0,C 180,E1 30408.289,E2 30408.289} C_VEL
LIN {X 0,Y 300.448,Z 1022.256,A -85,B 0,C 180,E1 30414.219,E2 30414.219} C_VEL
LIN {X 0,Y 300.366,Z 1024.681,A -85,B 0,C 180,E1 30418.165,E2 30418.165} C_VEL
LIN {X 0,Y 299.022,Z 1029.741,A -85,B 0,C 180,E1 30421.877,E2 30421.877} C_VEL
LIN {X 0,Y 264.872,Z 1067.265,A -85,B 0,C 180,E1 30425.375,E2 30425.375} C_VEL
LIN {X 0,Y 227.167,Z 1100.924,A -85,B 0,C 180,E1 30430.525,E2 30430.525} C_VEL
LIN {X 0,Y 192.127,Z 1127.209,A -85,B 0,C 180,E1 30437.503,E2 30437.503} C_VEL
LIN {X 0,Y 155.868,Z 1150.696,A -85,B 0,C 180,E1 30449.239,E2 30449.239} C_VEL
LIN {X 0,Y 129.529,Z 1166.614,A -85,B 0,C 180,E1 30465.57,E2 30465.57} C_VEL
LIN {X 0,Y 116.687,Z 1175.5,A -85,B 0,C 180,E1 30483.047,E2 30483.047} C_VEL
LIN {X 0,Y 112.615,Z 1180.452,A -85,B 0,C 180,E1 30502.285,E2 30502.285} C_VEL
LIN {X 0,Y 113.129,Z 1181.386,A -85,B 0,C 180,E1 30509.996,E2 30509.996} C_VEL
LIN {X 0,Y 113.06,Z 1180.953,A -85,B 0,C 180,E1 30525.501,E2 30525.501} C_VEL
LIN {X 0,Y 123.297,Z 1176.153,A -85,B 0,C 180,E1 30547.788,E2 30547.788} C_VEL
LIN {X 0,Y 148.751,Z 1165.193,A -85,B 0,C 180,E1 30566.934,E2 30566.934} C_VEL
LIN {X 0,Y 184.939,Z 1148.495,A -85,B 0,C 180,E1 30579.987,E2 30579.987} C_VEL
LIN {X 0,Y 226.872,Z 1125.367,A -85,B 0,C 180,E1 30588.484,E2 30588.484} C_VEL
LIN {X 0,Y 265.967,Z 1099.494,A -85,B 0,C 180,E1 30593.57,E2 30593.57} C_VEL
LIN {X 0,Y 305.885,Z 1067.286,A -85,B 0,C 180,E1 30597.176,E2 30597.176} C_VEL
LIN {X 0,Y 315.999,Z 1057.965,A -85,B 0,C 180,E1 30598.002,E2 30598.002} C_VEL
LIN {X 0,Y 313.74,Z 1059.938,A -85,B 0,C 180,E1 30598.49,E2 30598.49} C_VEL
LIN {X 0,Y 278.061,Z 1088.607,A -85,B 0,C 180,E1 30601.715,E2 30601.715} C_VEL
LIN {X 0,Y 237.183,Z 1115.048,A -85,B 0,C 180,E1 30606.755,E2 30606.755} C_VEL
LIN {X 0,Y 198.414,Z 1134.946,A -85,B 0,C 180,E1 30613.83,E2 30613.83} C_VEL
LIN {X 0,Y 161.992,Z 1149.876,A -85,B 0,C 180,E1 30624.636,E2 30624.636} C_VEL
LIN {X 0,Y 131.681,Z 1159.455,A -85,B 0,C 180,E1 30641.767,E2 30641.767} C_VEL
LIN {X 0,Y 117.629,Z 1162.822,A -85,B 0,C 180,E1 30659.083,E2 30659.083} C_VEL
LIN {X 0,Y 112.918,Z 1163.202,A -85,B 0,C 180,E1 30674.479,E2 30674.479} C_VEL
LIN {X 0,Y 113.704,Z 1161.61,A -85,B 0,C 180,E1 30690.004,E2 30690.004} C_VEL
LIN {X 0,Y 120.772,Z 1156.98,A -85,B 0,C 180,E1 30708.232,E2 30708.232} C_VEL
LIN {X 0,Y 138.857,Z 1147.313,A -85,B 0,C 180,E1 30726.77,E2 30726.77} C_VEL
LIN {X 0,Y 168.61,Z 1131.372,A -85,B 0,C 180,E1 30741.125,E2 30741.125} C_VEL
LIN {X 0,Y 183.601,Z 1122.602,A -85,B 0,C 180,E1 30745.864,E2 30745.864} C_VEL
LIN {X 0,Y 193.139,Z 1115.882,A -85,B 0,C 180,E1 30749.84,E2 30749.84} C_VEL
LIN {X 0,Y 203.181,Z 1108.63,A -85,B 0,C 180,E1 30753.432,E2 30753.432} C_VEL
LIN {X 0,Y 238.321,Z 1082.992,A -85,B 0,C 180,E1 30759.275,E2 30759.275} C_VEL
LIN {X 0,Y 275.553,Z 1049.5,A -85,B 0,C 180,E1 30763.684,E2 30763.684} C_VEL
LIN {X 0,Y 290.798,Z 1033.512,A -85,B 0,C 180,E1 30765.238,E2 30765.238} C_VEL
LIN {X 0,Y 292.829,Z 1030.151,A -85,B 0,C 180,E1 30768.669,E2 30768.669} C_VEL
LIN {X 0,Y 295.109,Z 1028.173,A -85,B 0,C 180,E1 30774.114,E2 30774.114} C_VEL
LIN {X 0,Y 295.291,Z 1029.503,A -85,B 0,C 180,E1 30777.058,E2 30777.058} C_VEL
LIN {X 0,Y 294.141,Z 1033.607,A -85,B 0,C 180,E1 30780.474,E2 30780.474} C_VEL
LIN {X 0,Y 291.676,Z 1036.814,A -85,B 0,C 180,E1 30780.965,E2 30780.965} C_VEL
LIN {X 0,Y 257.609,Z 1072.086,A -85,B 0,C 180,E1 30784.255,E2 30784.255} C_VEL
LIN {X 0,Y 221.851,Z 1102.889,A -85,B 0,C 180,E1 30788.997,E2 30788.997} C_VEL
LIN {X 0,Y 185.713,Z 1128.785,A -85,B 0,C 180,E1 30795.987,E2 30795.987} C_VEL
LIN {X 0,Y 151.935,Z 1149.731,A -85,B 0,C 180,E1 30806.468,E2 30806.468} C_VEL
LIN {X 0,Y 123.712,Z 1165.762,A -85,B 0,C 180,E1 30822.866,E2 30822.866} C_VEL
LIN {X 0,Y 109.471,Z 1174.728,A -85,B 0,C 180,E1 30841.105,E2 30841.105} C_VEL
LIN {X 0,Y 104.739,Z 1179.757,A -85,B 0,C 180,E1 30861.701,E2 30861.701} C_VEL
LIN {X 0,Y 105.235,Z 1180.723,A -85,B 0,C 180,E1 30869.996,E2 30869.996} C_VEL
LIN {X 0,Y 105.33,Z 1180.302,A -85,B 0,C 180,E1 30886.67,E2 30886.67} C_VEL
LIN {X 0,Y 116.888,Z 1175.539,A -85,B 0,C 180,E1 30910.266,E2 30910.266} C_VEL
LIN {X 0,Y 144.344,Z 1164.651,A -85,B 0,C 180,E1 30929.727,E2 30929.727} C_VEL
LIN {X 0,Y 181.955,Z 1148.162,A -85,B 0,C 180,E1 30942.398,E2 30942.398} C_VEL
LIN {X 0,Y 224.53,Z 1125.461,A -85,B 0,C 180,E1 30950.44,E2 30950.44} C_VEL
LIN {X 0,Y 266.233,Z 1098.433,A -85,B 0,C 180,E1 30955.448,E2 30955.448} C_VEL
LIN {X 0,Y 298.122,Z 1073.565,A -85,B 0,C 180,E1 30958.192,E2 30958.192} C_VEL
LIN {X 0,Y 260.107,Z 1100.969,A -85,B 0,C 180,E1 30961.803,E2 30961.803} C_VEL
LIN {X 0,Y 220.756,Z 1123.793,A -85,B 0,C 180,E1 30967.026,E2 30967.026} C_VEL
LIN {X 0,Y 181.496,Z 1141.776,A -85,B 0,C 180,E1 30974.913,E2 30974.913} C_VEL
LIN {X 0,Y 144.712,Z 1154.92,A -85,B 0,C 180,E1 30987.652,E2 30987.652} C_VEL
LIN {X 0,Y 122.422,Z 1161.086,A -85,B 0,C 180,E1 31002.221,E2 31002.221} C_VEL
LIN {X 0,Y 107.176,Z 1163.894,A -85,B 0,C 180,E1 31024.981,E2 31024.981} C_VEL
LIN {X 0,Y 104.765,Z 1163.398,A -85,B 0,C 180,E1 31041.711,E2 31041.711} C_VEL
LIN {X 0,Y 108.003,Z 1160.79,A -85,B 0,C 180,E1 31058.047,E2 31058.047} C_VEL
LIN {X 0,Y 119.531,Z 1154.525,A -85,B 0,C 180,E1 31077.709,E2 31077.709} C_VEL
LIN {X 0,Y 143.861,Z 1142.684,A -85,B 0,C 180,E1 31095.16,E2 31095.16} C_VEL
LIN {X 0,Y 178.872,Z 1123.839,A -85,B 0,C 180,E1 31107.815,E2 31107.815} C_VEL
LIN {X 0,Y 203.181,Z 1108.63,A -85,B 0,C 180,E1 31113.432,E2 31113.432} C_VEL
LIN {X 0,Y 213.751,Z 1100.942,A -85,B 0,C 180,E1 31116.66,E2 31116.66} C_VEL
LIN {X 0,Y 224.605,Z 1092.557,A -85,B 0,C 180,E1 31119.509,E2 31119.509} C_VEL
LIN {X 0,Y 261.322,Z 1062.372,A -85,B 0,C 180,E1 31124.027,E2 31124.027} C_VEL
LIN {X 0,Y 285.604,Z 1038.385,A -85,B 0,C 180,E1 31126.389,E2 31126.389} C_VEL
LIN {X 0,Y 288.524,Z 1034.844,A -85,B 0,C 180,E1 31130.951,E2 31130.951} C_VEL
LIN {X 0,Y 289.752,Z 1034.104,A -85,B 0,C 180,E1 31134.004,E2 31134.004} C_VEL
LIN {X 0,Y 289.936,Z 1035.413,A -85,B 0,C 180,E1 31137.004,E2 31137.004} C_VEL
LIN {X 0,Y 289.124,Z 1038.064,A -85,B 0,C 180,E1 31139.319,E2 31139.319} C_VEL
LIN {X 0,Y 280.362,Z 1047.656,A -85,B 0,C 180,E1 31140.215,E2 31140.215} C_VEL
LIN {X 0,Y 246.868,Z 1080.149,A -85,B 0,C 180,E1 31143.5,E2 31143.5} C_VEL
LIN {X 0,Y 208.678,Z 1110.622,A -85,B 0,C 180,E1 31148.717,E2 31148.717} C_VEL
LIN {X 0,Y 172.892,Z 1134.485,A -85,B 0,C 180,E1 31155.955,E2 31155.955} C_VEL
LIN {X 0,Y 135.227,Z 1155.93,A -85,B 0,C 180,E1 31169.25,E2 31169.25} C_VEL
LIN {X 0,Y 110.692,Z 1169.048,A -85,B 0,C 180,E1 31186.949,E2 31186.949} C_VEL
LIN {X 0,Y 99.73,Z 1175.985,A -85,B 0,C 180,E1 31205.33,E2 31205.33} C_VEL
LIN {X 0,Y 96.845,Z 1179.058,A -85,B 0,C 180,E1 31221.019,E2 31221.019} C_VEL
LIN {X 0,Y 97.316,Z 1180.056,A -85,B 0,C 180,E1 31229.996,E2 31229.996} C_VEL
LIN {X 0,Y 97.629,Z 1179.649,A -85,B 0,C 180,E1 31248.028,E2 31248.028} C_VEL
LIN {X 0,Y 110.7,Z 1174.924,A -85,B 0,C 180,E1 31273.037,E2 31273.037} C_VEL
LIN {X 0,Y 140.248,Z 1164.135,A -85,B 0,C 180,E1 31292.66,E2 31292.66} C_VEL
LIN {X 0,Y 180.339,Z 1147.353,A -85,B 0,C 180,E1 31305.128,E2 31305.128} C_VEL
LIN {X 0,Y 226.008,Z 1123.535,A -85,B 0,C 180,E1 31312.913,E2 31312.913} C_VEL
LIN {X 0,Y 267.111,Z 1097.135,A -85,B 0,C 180,E1 31317.345,E2 31317.345} C_VEL
LIN {X 0,Y 277.233,Z 1089.726,A -85,B 0,C 180,E1 31318.332,E2 31318.332} C_VEL
LIN {X 0,Y 234.507,Z 1116.451,A -85,B 0,C 180,E1 31322.85,E2 31322.85} C_VEL
LIN {X 0,Y 192.859,Z 1136.745,A -85,B 0,C 180,E1 31329.419,E2 31329.419} C_VEL
LIN {X 0,Y 152.996,Z 1151.772,A -85,B 0,C 180,E1 31339.881,E2 31339.881} C_VEL
LIN {X 0,Y 121.119,Z 1160.618,A -85,B 0,C 180,E1 31355.816,E2 31355.816} C_VEL
LIN {X 0,Y 103.829,Z 1164.084,A -85,B 0,C 180,E1 31374.402,E2 31374.402} C_VEL
LIN {X 0,Y 97.479,Z 1164.563,A -85,B 0,C 180,E1 31391.943,E2 31391.943} C_VEL
LIN {X 0,Y 97.829,Z 1163.007,A -85,B 0,C 180,E1 31410.004,E2 31410.004} C_VEL
LIN {X 0,Y 103.692,Z 1159.621,A -85,B 0,C 180,E1 31426.95,E2 31426.95} C_VEL
LIN {X 0,Y 122.38,Z 1150.891,A -85,B 0,C 180,E1 31448.13,E2 31448.13} C_VEL
LIN {X 0,Y 153.23,Z 1136.317,A -85,B 0,C 180,E1 31463.527,E2 31463.527} C_VEL
LIN {X 0,Y 189.669,Z 1116.091,A -85,B 0,C 180,E1 31473.456,E2 31473.456} C_VEL
LIN {X 0,Y 224.605,Z 1092.557,A -85,B 0,C 180,E1 31479.509,E2 31479.509} C_VEL
LIN {X 0,Y 235.603,Z 1083.837,A -85,B 0,C 180,E1 31482.092,E2 31482.092} C_VEL
LIN {X 0,Y 246.824,Z 1074.442,A -85,B 0,C 180,E1 31484.42,E2 31484.42} C_VEL
LIN {X 0,Y 281.085,Z 1042.646,A -85,B 0,C 180,E1 31487.786,E2 31487.786} C_VEL
LIN {X 0,Y 282.826,Z 1040.691,A -85,B 0,C 180,E1 31490.768,E2 31490.768} C_VEL
LIN {X 0,Y 284.23,Z 1039.919,A -85,B 0,C 180,E1 31493.988,E2 31493.988} C_VEL
LIN {X 0,Y 283.918,Z 1042.445,A -85,B 0,C 180,E1 31498.155,E2 31498.155} C_VEL
LIN {X 0,Y 247.794,Z 1077.747,A -85,B 0,C 180,E1 31501.41,E2 31501.41} C_VEL
LIN {X 0,Y 209.93,Z 1107.737,A -85,B 0,C 180,E1 31506.028,E2 31506.028} C_VEL
LIN {X 0,Y 170.755,Z 1133.465,A -85,B 0,C 180,E1 31513.217,E2 31513.217} C_VEL
LIN {X 0,Y 131.399,Z 1154.954,A -85,B 0,C 180,E1 31525.997,E2 31525.997} C_VEL
LIN {X 0,Y 104.772,Z 1168.233,A -85,B 0,C 180,E1 31543.844,E2 31543.844} C_VEL
LIN {X 0,Y 92.129,Z 1175.429,A -85,B 0,C 180,E1 31563.997,E2 31563.997} C_VEL
LIN {X 0,Y 88.979,Z 1178.359,A -85,B 0,C 180,E1 31580.217,E2 31580.217} C_VEL
LIN {X 0,Y 89.393,Z 1179.39,A -85,B 0,C 180,E1 31589.995,E2 31589.995} C_VEL
LIN {X 0,Y 90.019,Z 1178.999,A -85,B 0,C 180,E1 31609.612,E2 31609.612} C_VEL
LIN {X 0,Y 104.794,Z 1174.307,A -85,B 0,C 180,E1 31636.131,E2 31636.131} C_VEL
LIN {X 0,Y 133.797,Z 1164.645,A -85,B 0,C 180,E1 31654.619,E2 31654.619} C_VEL
LIN {X 0,Y 175.583,Z 1148.06,A -85,B 0,C 180,E1 31667.145,E2 31667.145} C_VEL
LIN {X 0,Y 219.176,Z 1126.49,A -85,B 0,C 180,E1 31674.278,E2 31674.278} C_VEL
LIN {X 0,Y 256.984,Z 1103.52,A -85,B 0,C 180,E1 31678.403,E2 31678.403} C_VEL
LIN {X 0,Y 215.35,Z 1126.572,A -85,B 0,C 180,E1 31683.183,E2 31683.183} C_VEL
LIN {X 0,Y 173.238,Z 1144.424,A -85,B 0,C 180,E1 31690.645,E2 31690.645} C_VEL
LIN {X 0,Y 137.874,Z 1155.912,A -85,B 0,C 180,E1 31701.32,E2 31701.32} C_VEL
LIN {X 0,Y 111.816,Z 1162.25,A -85,B 0,C 180,E1 31715.826,E2 31715.826} C_VEL
LIN {X 0,Y 92.605,Z 1165.212,A -85,B 0,C 180,E1 31740.695,E2 31740.695} C_VEL
LIN {X 0,Y 88.917,Z 1164.751,A -85,B 0,C 180,E1 31760.22,E2 31760.22} C_VEL
LIN {X 0,Y 92.402,Z 1162.244,A -85,B 0,C 180,E1 31779.417,E2 31779.417} C_VEL
LIN {X 0,Y 104.317,Z 1156.762,A -85,B 0,C 180,E1 31799.989,E2 31799.989} C_VEL
LIN {X 0,Y 133.252,Z 1144.475,A -85,B 0,C 180,E1 31819.954,E2 31819.954} C_VEL
LIN {X 0,Y 170.818,Z 1125.891,A -85,B 0,C 180,E1 31832.213,E2 31832.213} C_VEL
LIN {X 0,Y 207.883,Z 1103.492,A -85,B 0,C 180,E1 31839.38,E2 31839.38} C_VEL
LIN {X 0,Y 246.824,Z 1074.442,A -85,B 0,C 180,E1 31844.42,E2 31844.42} C_VEL
LIN {X 0,Y 258.09,Z 1064.603,A -85,B 0,C 180,E1 31846.513,E2 31846.513} C_VEL
LIN {X 0,Y 269.202,Z 1054.139,A -85,B 0,C 180,E1 31848.392,E2 31848.392} C_VEL
LIN {X 0,Y 274.555,Z 1049.116,A -85,B 0,C 180,E1 31848.811,E2 31848.811} C_VEL
LIN {X 0,Y 276.551,Z 1047.078,A -85,B 0,C 180,E1 31849.603,E2 31849.603} C_VEL
LIN {X 0,Y 278.595,Z 1045.653,A -85,B 0,C 180,E1 31853.971,E2 31853.971} C_VEL
LIN {X 0,Y 278.746,Z 1046.855,A -85,B 0,C 180,E1 31856.884,E2 31856.884} C_VEL
LIN {X 0,Y 243.485,Z 1080.041,A -85,B 0,C 180,E1 31859.854,E2 31859.854} C_VEL
LIN {X 0,Y 203.517,Z 1110.612,A -85,B 0,C 180,E1 31864.505,E2 31864.505} C_VEL
LIN {X 0,Y 165.587,Z 1134.337,A -85,B 0,C 180,E1 31871.164,E2 31871.164} C_VEL
LIN {X 0,Y 126.061,Z 1154.972,A -85,B 0,C 180,E1 31883.416,E2 31883.416} C_VEL
LIN {X 0,Y 96.767,Z 1168.495,A -85,B 0,C 180,E1 31902.834,E2 31902.834} C_VEL
LIN {X 0,Y 82.71,Z 1176.014,A -85,B 0,C 180,E1 31928.562,E2 31928.562} C_VEL
LIN {X 0,Y 81.464,Z 1178.724,A -85,B 0,C 180,E1 31949.995,E2 31949.995} C_VEL
LIN {X 0,Y 83.398,Z 1178.105,A -85,B 0,C 180,E1 31975.111,E2 31975.111} C_VEL
LIN {X 0,Y 99.226,Z 1173.691,A -85,B 0,C 180,E1 31999.586,E2 31999.586} C_VEL
LIN {X 0,Y 130.42,Z 1164.11,A -85,B 0,C 180,E1 32017.953,E2 32017.953} C_VEL
LIN {X 0,Y 175.132,Z 1147.077,A -85,B 0,C 180,E1 32030.076,E2 32030.076} C_VEL
LIN {X 0,Y 220.166,Z 1125.198,A -85,B 0,C 180,E1 32036.656,E2 32036.656} C_VEL
LIN {X 0,Y 236.699,Z 1115.825,A -85,B 0,C 180,E1 32038.364,E2 32038.364} C_VEL
LIN {X 0,Y 196.795,Z 1135.215,A -85,B 0,C 180,E1 32043.449,E2 32043.449} C_VEL
LIN {X 0,Y 151.087,Z 1151.839,A -85,B 0,C 180,E1 32052.809,E2 32052.809} C_VEL
LIN {X 0,Y 117.413,Z 1160.746,A -85,B 0,C 180,E1 32065.731,E2 32065.731} C_VEL
LIN {X 0,Y 90.891,Z 1165.354,A -85,B 0,C 180,E1 32088.322,E2 32088.322} C_VEL
LIN {X 0,Y 82.269,Z 1165.927,A -85,B 0,C 180,E1 32108.453,E2 32108.453} C_VEL
LIN {X 0,Y 81.912,Z 1164.41,A -85,B 0,C 180,E1 32130.005,E2 32130.005} C_VEL
LIN {X 0,Y 88.796,Z 1161.133,A -85,B 0,C 180,E1 32149.904,E2 32149.904} C_VEL
LIN {X 0,Y 110.444,Z 1152.538,A -85,B 0,C 180,E1 32173.172,E2 32173.172} C_VEL
LIN {X 0,Y 142.895,Z 1138.926,A -85,B 0,C 180,E1 32188.058,E2 32188.058} C_VEL
LIN {X 0,Y 184.568,Z 1117.333,A -85,B 0,C 180,E1 32198.087,E2 32198.087} C_VEL
LIN {X 0,Y 223.81,Z 1091.777,A -85,B 0,C 180,E1 32203.874,E2 32203.874} C_VEL
LIN {X 0,Y 261.034,Z 1061.811,A -85,B 0,C 180,E1 32207.667,E2 32207.667} C_VEL
LIN {X 0,Y 269.202,Z 1054.139,A -85,B 0,C 180,E1 32208.392,E2 32208.392} C_VEL
LIN {X 0,Y 271.971,Z 1051.507,A -85,B 0,C 180,E1 32209.337,E2 32209.337} C_VEL
LIN {X 0,Y 272.71,Z 1051.324,A -85,B 0,C 180,E1 32213.313,E2 32213.313} C_VEL
LIN {X 0,Y 272.805,Z 1052.094,A -85,B 0,C 180,E1 32215.627,E2 32215.627} C_VEL
LIN {X 0,Y 232.136,Z 1088.149,A -85,B 0,C 180,E1 32218.872,E2 32218.872} C_VEL
LIN {X 0,Y 191.817,Z 1116.803,A -85,B 0,C 180,E1 32223.625,E2 32223.625} C_VEL
LIN {X 0,Y 150.907,Z 1140.497,A -85,B 0,C 180,E1 32231.184,E2 32231.184} C_VEL
LIN {X 0,Y 112.194,Z 1158.769,A -85,B 0,C 180,E1 32244.602,E2 32244.602} C_VEL
LIN {X 0,Y 85.743,Z 1170.126,A -85,B 0,C 180,E1 32265.167,E2 32265.167} C_VEL
LIN {X 0,Y 75.257,Z 1175.281,A -85,B 0,C 180,E1 32286.316,E2 32286.316} C_VEL
LIN {X 0,Y 73.532,Z 1178.056,A -85,B 0,C 180,E1 32309.994,E2 32309.994} C_VEL
LIN {X 0,Y 74.991,Z 1177.693,A -85,B 0,C 180,E1 32333.76,E2 32333.76} C_VEL
LIN {X 0,Y 94.061,Z 1173.077,A -85,B 0,C 180,E1 32363.436,E2 32363.436} C_VEL
LIN {X 0,Y 127.512,Z 1163.577,A -85,B 0,C 180,E1 32381.444,E2 32381.444} C_VEL
LIN {X 0,Y 173.878,Z 1146.603,A -85,B 0,C 180,E1 32392.813,E2 32392.813} C_VEL
LIN {X 0,Y 216.249,Z 1126.747,A -85,B 0,C 180,E1 32398.553,E2 32398.553} C_VEL
LIN {X 0,Y 175.703,Z 1143.691,A -85,B 0,C 180,E1 32404.201,E2 32404.201} C_VEL
LIN {X 0,Y 132.342,Z 1157.05,A -85,B 0,C 180,E1 32414.583,E2 32414.583} C_VEL
LIN {X 0,Y 102.866,Z 1163.421,A -85,B 0,C 180,E1 32428.196,E2 32428.196} C_VEL
LIN {X 0,Y 78.709,Z 1166.534,A -85,B 0,C 180,E1 32454.839,E2 32454.839} C_VEL
LIN {X 0,Y 73.137,Z 1166.104,A -85,B 0,C 180,E1 32478.082,E2 32478.082} C_VEL
LIN {X 0,Y 76.873,Z 1163.7,A -85,B 0,C 180,E1 32501.342,E2 32501.342} C_VEL
LIN {X 0,Y 91.459,Z 1158.191,A -85,B 0,C 180,E1 32525.336,E2 32525.336} C_VEL
LIN {X 0,Y 123.724,Z 1146.221,A -85,B 0,C 180,E1 32545.536,E2 32545.536} C_VEL
LIN {X 0,Y 164.084,Z 1127.818,A -85,B 0,C 180,E1 32557.072,E2 32557.072} C_VEL
LIN {X 0,Y 202.901,Z 1105.682,A -85,B 0,C 180,E1 32563.52,E2 32563.52} C_VEL
LIN {X 0,Y 243.342,Z 1076.645,A -85,B 0,C 180,E1 32567.984,E2 32567.984} C_VEL
LIN {X 0,Y 271.25,Z 1052.195,A -85,B 0,C 180,E1 32570.37,E2 32570.37} C_VEL
LIN {X 0,Y 272.71,Z 1051.324,A -85,B 0,C 180,E1 32573.313,E2 32573.313} C_VEL
LIN {X 0,Y 270.571,Z 1053.642,A -85,B 0,C 180,E1 32574.261,E2 32574.261} C_VEL
LIN {X 0,Y 261.855,Z 1061.912,A -85,B 0,C 180,E1 32574.784,E2 32574.784} C_VEL
LIN {X 0,Y 256.473,Z 1066.727,A -85,B 0,C 180,E1 32575.002,E2 32575.002} C_VEL
LIN {X 0,Y 216.033,Z 1099.231,A -85,B 0,C 180,E1 32578.324,E2 32578.324} C_VEL
LIN {X 0,Y 174.116,Z 1126.134,A -85,B 0,C 180,E1 32583.521,E2 32583.521} C_VEL
LIN {X 0,Y 132.538,Z 1147.698,A -85,B 0,C 180,E1 32592.212,E2 32592.212} C_VEL
LIN {X 0,Y 94.017,Z 1163.86,A -85,B 0,C 180,E1 32608.8,E2 32608.8} C_VEL
LIN {X 0,Y 72.839,Z 1172.227,A -85,B 0,C 180,E1 32631.502,E2 32631.502} C_VEL
LIN {X 0,Y 65.442,Z 1176.26,A -85,B 0,C 180,E1 32656.642,E2 32656.642} C_VEL
LIN {X 0,Y 65.619,Z 1177.379,A -85,B 0,C 180,E1 32669.993,E2 32669.993} C_VEL
LIN {X 0,Y 67.807,Z 1177.012,A -85,B 0,C 180,E1 32697.022,E2 32697.022} C_VEL
LIN {X 0,Y 89.366,Z 1172.463,A -85,B 0,C 180,E1 32727.714,E2 32727.714} C_VEL
LIN {X 0,Y 125.095,Z 1163.043,A -85,B 0,C 180,E1 32745.09,E2 32745.09} C_VEL
LIN {X 0,Y 174.709,Z 1145.475,A -85,B 0,C 180,E1 32755.826,E2 32755.826} C_VEL
LIN {X 0,Y 195.77,Z 1136.385,A -85,B 0,C 180,E1 32758.548,E2 32758.548} C_VEL
LIN {X 0,Y 147.914,Z 1152.935,A -85,B 0,C 180,E1 32766.484,E2 32766.484} C_VEL
LIN {X 0,Y 105.391,Z 1162.897,A -85,B 0,C 180,E1 32780.522,E2 32780.522} C_VEL
LIN {X 0,Y 79.268,Z 1166.63,A -85,B 0,C 180,E1 32800.32,E2 32800.32} C_VEL
LIN {X 0,Y 67.288,Z 1167.267,A -85,B 0,C 180,E1 32824.02,E2 32824.02} C_VEL
LIN {X 0,Y 65.989,Z 1165.815,A -85,B 0,C 180,E1 32850.007,E2 32850.007} C_VEL
LIN {X 0,Y 74.231,Z 1162.64,A -85,B 0,C 180,E1 32874.032,E2 32874.032} C_VEL
LIN {X 0,Y 99.553,Z 1154.177,A -85,B 0,C 180,E1 32899.379,E2 32899.379} C_VEL
LIN {X 0,Y 138.156,Z 1139.463,A -85,B 0,C 180,E1 32914.479,E2 32914.479} C_VEL
LIN {X 0,Y 180.81,Z 1118.534,A -85,B 0,C 180,E1 32922.971,E2 32922.971} C_VEL
LIN {X 0,Y 220.376,Z 1093.783,A -85,B 0,C 180,E1 32927.839,E2 32927.839} C_VEL
LIN {X 0,Y 259.974,Z 1062.762,A -85,B 0,C 180,E1 32931.179,E2 32931.179} C_VEL
LIN {X 0,Y 266.044,Z 1057.201,A -85,B 0,C 180,E1 32931.787,E2 32931.787} C_VEL
LIN {X 0,Y 267.144,Z 1056.726,A -85,B 0,C 180,E1 32934.024,E2 32934.024} C_VEL
LIN {X 0,Y 261.851,Z 1061.865,A -85,B 0,C 180,E1 32934.647,E2 32934.647} C_VEL
LIN {X 0,Y 256.473,Z 1066.727,A -85,B 0,C 180,E1 32935.002,E2 32935.002} C_VEL
LIN {X 0,Y 243.01,Z 1078.006,A -85,B 0,C 180,E1 32935.011,E2 32935.011} C_VEL
LIN {X 0,Y 229.109,Z 1088.706,A -85,B 0,C 180,E1 32935.014,E2 32935.014} C_VEL
LIN {X 0,Y 185.135,Z 1118.489,A -85,B 0,C 180,E1 32939.275,E2 32939.275} C_VEL
LIN {X 0,Y 143.722,Z 1140.779,A -85,B 0,C 180,E1 32945.714,E2 32945.714} C_VEL
LIN {X 0,Y 101.22,Z 1158.998,A -85,B 0,C 180,E1 32958.488,E2 32958.488} C_VEL
LIN {X 0,Y 69.617,Z 1170.365,A -85,B 0,C 180,E1 32982.559,E2 32982.559} C_VEL
LIN {X 0,Y 57.677,Z 1175.558,A -85,B 0,C 180,E1 33014.804,E2 33014.804} C_VEL
LIN {X 0,Y 57.682,Z 1176.687,A -85,B 0,C 180,E1 33029.993,E2 33029.993} C_VEL
LIN {X 0,Y 60.519,Z 1176.384,A -85,B 0,C 180,E1 33059.951,E2 33059.951} C_VEL
LIN {X 0,Y 79.857,Z 1172.93,A -85,B 0,C 180,E1 33088.368,E2 33088.368} C_VEL
LIN {X 0,Y 116.398,Z 1164.333,A -85,B 0,C 180,E1 33106.809,E2 33106.809} C_VEL
LIN {X 0,Y 162.674,Z 1149.492,A -85,B 0,C 180,E1 33116.917,E2 33116.917} C_VEL
LIN {X 0,Y 174.424,Z 1144.922,A -85,B 0,C 180,E1 33118.782,E2 33118.782} C_VEL
LIN {X 0,Y 127.087,Z 1158.616,A -85,B 0,C 180,E1 33127.821,E2 33127.821} C_VEL
LIN {X 0,Y 96.055,Z 1164.592,A -85,B 0,C 180,E1 33139.294,E2 33139.294} C_VEL
LIN {X 0,Y 65.93,Z 1167.862,A -85,B 0,C 180,E1 33166.568,E2 33166.568} C_VEL
LIN {X 0,Y 57.505,Z 1167.458,A -85,B 0,C 180,E1 33194.773,E2 33194.773} C_VEL
LIN {X 0,Y 61.468,Z 1165.152,A -85,B 0,C 180,E1 33224.239,E2 33224.239} C_VEL
LIN {X 0,Y 79.145,Z 1159.764,A -85,B 0,C 180,E1 33251.941,E2 33251.941} C_VEL
LIN {X 0,Y 115.556,Z 1147.924,A -85,B 0,C 180,E1 33271.977,E2 33271.977} C_VEL
LIN {X 0,Y 155.191,Z 1131.388,A -85,B 0,C 180,E1 33281.701,E2 33281.701} C_VEL
LIN {X 0,Y 199.028,Z 1107.865,A -85,B 0,C 180,E1 33287.844,E2 33287.844} C_VEL
LIN {X 0,Y 240.577,Z 1079.015,A -85,B 0,C 180,E1 33291.623,E2 33291.623} C_VEL
LIN {X 0,Y 258.799,Z 1064.129,A -85,B 0,C 180,E1 33293.053,E2 33293.053} C_VEL
LIN {X 0,Y 229.109,Z 1088.706,A -85,B 0,C 180,E1 33295.014,E2 33295.014} C_VEL
LIN {X 0,Y 214.668,Z 1098.91,A -85,B 0,C 180,E1 33295.075,E2 33295.075} C_VEL
LIN {X 0,Y 200.044,Z 1108.359,A -85,B 0,C 180,E1 33295.24,E2 33295.24} C_VEL
LIN {X 0,Y 158.002,Z 1132.492,A -85,B 0,C 180,E1 33299.985,E2 33299.985} C_VEL
LIN {X 0,Y 113.849,Z 1152.466,A -85,B 0,C 180,E1 33308.883,E2 33308.883} C_VEL
LIN {X 0,Y 75.828,Z 1165.911,A -85,B 0,C 180,E1 33326.25,E2 33326.25} C_VEL
LIN {X 0,Y 52.855,Z 1173.452,A -85,B 0,C 180,E1 33358.975,E2 33358.975} C_VEL
LIN {X 0,Y 49.756,Z 1175.991,A -85,B 0,C 180,E1 33389.991,E2 33389.991} C_VEL
LIN {X 0,Y 53.629,Z 1175.727,A -85,B 0,C 180,E1 33424.292,E2 33424.292} C_VEL
LIN {X 0,Y 81.705,Z 1171.233,A -85,B 0,C 180,E1 33457.616,E2 33457.616} C_VEL
LIN {X 0,Y 122.813,Z 1161.698,A -85,B 0,C 180,E1 33472.952,E2 33472.952} C_VEL
LIN {X 0,Y 153.986,Z 1151.963,A -85,B 0,C 180,E1 33478.797,E2 33478.797} C_VEL
LIN {X 0,Y 107.162,Z 1163.027,A -85,B 0,C 180,E1 33489.239,E2 33489.239} C_VEL
LIN {X 0,Y 69.664,Z 1167.909,A -85,B 0,C 180,E1 33509.824,E2 33509.824} C_VEL
LIN {X 0,Y 51.58,Z 1168.463,A -85,B 0,C 180,E1 33541.61,E2 33541.61} C_VEL
LIN {X 0,Y 50.047,Z 1167.219,A -85,B 0,C 180,E1 33570.009,E2 33570.009} C_VEL
LIN {X 0,Y 60.244,Z 1164.145,A -85,B 0,C 180,E1 33600.119,E2 33600.119} C_VEL
LIN {X 0,Y 90.107,Z 1155.813,A -85,B 0,C 180,E1 33626.993,E2 33626.993} C_VEL
LIN {X 0,Y 132.153,Z 1141.312,A -85,B 0,C 180,E1 33640.634,E2 33640.634} C_VEL
LIN {X 0,Y 177.562,Z 1120.167,A -85,B 0,C 180,E1 33647.911,E2 33647.911} C_VEL
LIN {X 0,Y 217.99,Z 1095.789,A -85,B 0,C 180,E1 33651.903,E2 33651.903} C_VEL
LIN {X 0,Y 228.533,Z 1088.493,A -85,B 0,C 180,E1 33652.692,E2 33652.692} C_VEL
LIN {X 0,Y 227.485,Z 1089.322,A -85,B 0,C 180,E1 33653.08,E2 33653.08} C_VEL
LIN {X 0,Y 200.044,Z 1108.359,A -85,B 0,C 180,E1 33655.24,E2 33655.24} C_VEL
LIN {X 0,Y 192.659,Z 1112.953,A -85,B 0,C 180,E1 33655.548,E2 33655.548} C_VEL
LIN {X 0,Y 171.381,Z 1124.579,A -85,B 0,C 180,E1 33655.465,E2 33655.465} C_VEL
LIN {X 0,Y 169.512,Z 1125.586,A -85,B 0,C 180,E1 33655.642,E2 33655.642} C_VEL
LIN {X 0,Y 124.759,Z 1146.782,A -85,B 0,C 180,E1 33662.091,E2 33662.091} C_VEL
LIN {X 0,Y 78.867,Z 1163.225,A -85,B 0,C 180,E1 33676.642,E2 33676.642} C_VEL
LIN {X 0,Y 51.159,Z 1171.254,A -85,B 0,C 180,E1 33702.388,E2 33702.388} C_VEL
LIN {X 0,Y 42.414,Z 1174.153,A -85,B 0,C 180,E1 33729.117,E2 33729.117} C_VEL
LIN {X 0,Y 41.82,Z 1175.293,A -85,B 0,C 180,E1 33749.99,E2 33749.99} C_VEL
LIN {X 0,Y 47.129,Z 1175.071,A -85,B 0,C 180,E1 33789.875,E2 33789.875} C_VEL
LIN {X 0,Y 78.919,Z 1170.621,A -85,B 0,C 180,E1 33823.194,E2 33823.194} C_VEL
LIN {X 0,Y 125.862,Z 1160.079,A -85,B 0,C 180,E1 33837.58,E2 33837.58} C_VEL
LIN {X 0,Y 130.665,Z 1158.7,A -85,B 0,C 180,E1 33838.461,E2 33838.461} C_VEL
LIN {X 0,Y 126.59,Z 1159.523,A -85,B 0,C 180,E1 33840.019,E2 33840.019} C_VEL
LIN {X 0,Y 91.223,Z 1165.866,A -85,B 0,C 180,E1 33849.562,E2 33849.562} C_VEL
LIN {X 0,Y 55.121,Z 1169.192,A -85,B 0,C 180,E1 33874.683,E2 33874.683} C_VEL
LIN {X 0,Y 42.192,Z 1168.813,A -85,B 0,C 180,E1 33909.024,E2 33909.024} C_VEL
LIN {X 0,Y 46.299,Z 1166.607,A -85,B 0,C 180,E1 33949.059,E2 33949.059} C_VEL
LIN {X 0,Y 62.957,Z 1162.64,A -85,B 0,C 180,E1 33976.071,E2 33976.071} C_VEL
LIN {X 0,Y 102.346,Z 1151.775,A -85,B 0,C 180,E1 33997.351,E2 33997.351} C_VEL
LIN {X 0,Y 147.419,Z 1134.954,A -85,B 0,C 180,E1 34006.869,E2 34006.869} C_VEL
LIN {X 0,Y 192.662,Z 1112.042,A -85,B 0,C 180,E1 34012.002,E2 34012.002} C_VEL
LIN {X 0,Y 200.611,Z 1107.394,A -85,B 0,C 180,E1 34012.859,E2 34012.859} C_VEL
LIN {X 0,Y 169.512,Z 1125.586,A -85,B 0,C 180,E1 34015.642,E2 34015.642} C_VEL
LIN {X 0,Y 161.808,Z 1129.6,A -85,B 0,C 180,E1 34016.069,E2 34016.069} C_VEL
LIN {X 0,Y 139.675,Z 1139.478,A -85,B 0,C 180,E1 34016.083,E2 34016.083} C_VEL
LIN {X 0,Y 137.721,Z 1140.312,A -85,B 0,C 180,E1 34016.299,E2 34016.299} C_VEL
LIN {X 0,Y 91.104,Z 1158.054,A -85,B 0,C 180,E1 34025.564,E2 34025.564} C_VEL
LIN {X 0,Y 51.359,Z 1169.101,A -85,B 0,C 180,E1 34048.015,E2 34048.015} C_VEL
LIN {X 0,Y 35.009,Z 1173.447,A -85,B 0,C 180,E1 34084.414,E2 34084.414} C_VEL
LIN {X 0,Y 33.88,Z 1174.595,A -85,B 0,C 180,E1 34109.987,E2 34109.987} C_VEL
LIN {X 0,Y 41.225,Z 1174.416,A -85,B 0,C 180,E1 34157.132,E2 34157.132} C_VEL
LIN {X 0,Y 76.927,Z 1170.009,A -85,B 0,C 180,E1 34189.138,E2 34189.138} C_VEL
LIN {X 0,Y 111.332,Z 1163.127,A -85,B 0,C 180,E1 34198.963,E2 34198.963} C_VEL
LIN {X 0,Y 69.755,Z 1168.721,A -85,B 0,C 180,E1 34212.547,E2 34212.547} C_VEL
LIN {X 0,Y 40.943,Z 1169.93,A -85,B 0,C 180,E1 34242.44,E2 34242.44} C_VEL
LIN {X 0,Y 34.07,Z 1168.624,A -85,B 0,C 180,E1 34290.013,E2 34290.013} C_VEL
LIN {X 0,Y 47.331,Z 1165.646,A -85,B 0,C 180,E1 34329.695,E2 34329.695} C_VEL
LIN {X 0,Y 82.608,Z 1157.444,A -85,B 0,C 180,E1 34356.168,E2 34356.168} C_VEL
LIN {X 0,Y 127.803,Z 1143.128,A -85,B 0,C 180,E1 34367.299,E2 34367.299} C_VEL
LIN {X 0,Y 170.282,Z 1124.552,A -85,B 0,C 180,E1 34372.786,E2 34372.786} C_VEL
LIN {X 0,Y 137.721,Z 1140.312,A -85,B 0,C 180,E1 34376.299,E2 34376.299} C_VEL
LIN {X 0,Y 121.431,Z 1146.733,A -85,B 0,C 180,E1 34376.781,E2 34376.781} C_VEL
LIN {X 0,Y 104.859,Z 1152.444,A -85,B 0,C 180,E1 34377.378,E2 34377.378} C_VEL
LIN {X 0,Y 61.457,Z 1165.212,A -85,B 0,C 180,E1 34390.371,E2 34390.371} C_VEL
LIN {X 0,Y 36.344,Z 1170.836,A -85,B 0,C 180,E1 34413.719,E2 34413.719} C_VEL
LIN {X 0,Y 25.908,Z 1173.895,A -85,B 0,C 180,E1 34469.983,E2 34469.983} C_VEL
LIN {X 0,Y 36.172,Z 1173.758,A -85,B 0,C 180,E1 34526.65,E2 34526.65} C_VEL
LIN {X 0,Y 75.8,Z 1169.397,A -85,B 0,C 180,E1 34555.33,E2 34555.33} C_VEL
LIN {X 0,Y 88.505,Z 1167.297,A -85,B 0,C 180,E1 34558.821,E2 34558.821} C_VEL
LIN {X 0,Y 61.195,Z 1169.838,A -85,B 0,C 180,E1 34569.024,E2 34569.024} C_VEL
LIN {X 0,Y 35.912,Z 1170.593,A -85,B 0,C 180,E1 34592.716,E2 34592.716} C_VEL
LIN {X 0,Y 26.065,Z 1169.328,A -85,B 0,C 180,E1 34650.017,E2 34650.017} C_VEL
LIN {X 0,Y 41.594,Z 1166.378,A -85,B 0,C 180,E1 34696.618,E2 34696.618} C_VEL
LIN {X 0,Y 79.751,Z 1158.259,A -85,B 0,C 180,E1 34721.351,E2 34721.351} C_VEL
LIN {X 0,Y 127.561,Z 1143.567,A -85,B 0,C 180,E1 34730.949,E2 34730.949} C_VEL
LIN {X 0,Y 137.304,Z 1139.724,A -85,B 0,C 180,E1 34732.125,E2 34732.125} C_VEL
LIN {X 0,Y 137.042,Z 1139.959,A -85,B 0,C 180,E1 34732.962,E2 34732.962} C_VEL
LIN {X 0,Y 104.859,Z 1152.444,A -85,B 0,C 180,E1 34737.378,E2 34737.378} C_VEL
LIN {X 0,Y 88.089,Z 1157.509,A -85,B 0,C 180,E1 34738.191,E2 34738.191} C_VEL
LIN {X 0,Y 71.131,Z 1161.81,A -85,B 0,C 180,E1 34739.257,E2 34739.257} C_VEL
LIN {X 0,Y 32.524,Z 1170.091,A -85,B 0,C 180,E1 34761.649,E2 34761.649} C_VEL
LIN {X 0,Y 17.952,Z 1173.197,A -85,B 0,C 180,E1 34829.976,E2 34829.976} C_VEL
LIN {X 0,Y 32.412,Z 1173.101,A -85,B 0,C 180,E1 34898.782,E2 34898.782} C_VEL
LIN {X 0,Y 60.505,Z 1170.798,A -85,B 0,C 180,E1 34917.301,E2 34917.301} C_VEL
LIN {X 0,Y 63.688,Z 1170.333,A -85,B 0,C 180,E1 34920.038,E2 34920.038} C_VEL
LIN {X 0,Y 32.218,Z 1171.255,A -85,B 0,C 180,E1 34940.31,E2 34940.31} C_VEL
LIN {X 0,Y 18.052,Z 1170.033,A -85,B 0,C 180,E1 35010.024,E2 35010.024} C_VEL
LIN {X 0,Y 36.648,Z 1167.097,A -85,B 0,C 180,E1 35065.577,E2 35065.577} C_VEL
LIN {X 0,Y 77.597,Z 1159.072,A -85,B 0,C 180,E1 35086.855,E2 35086.855} C_VEL
LIN {X 0,Y 106.778,Z 1151.091,A -85,B 0,C 180,E1 35092.187,E2 35092.187} C_VEL
LIN {X 0,Y 102.243,Z 1152.624,A -85,B 0,C 180,E1 35093.252,E2 35093.252} C_VEL
LIN {X 0,Y 71.131,Z 1161.81,A -85,B 0,C 180,E1 35099.257,E2 35099.257} C_VEL
LIN {X 0,Y 54.083,Z 1165.466,A -85,B 0,C 180,E1 35100.778,E2 35100.778} C_VEL
LIN {X 0,Y 36.79,Z 1168.319,A -85,B 0,C 180,E1 35103.088,E2 35103.088} C_VEL
LIN {X 0,Y 16.824,Z 1171.298,A -85,B 0,C 180,E1 35126.021,E2 35126.021} C_VEL
LIN {X 0,Y 9.98,Z 1172.498,A -85,B 0,C 180,E1 35189.957,E2 35189.957} C_VEL
LIN {X 0,Y 30.423,Z 1172.442,A -85,B 0,C 180,E1 35273.288,E2 35273.288} C_VEL
LIN {X 0,Y 39.627,Z 1171.884,A -85,B 0,C 180,E1 35280.06,E2 35280.06} C_VEL
LIN {X 0,Y 16.637,Z 1171.544,A -85,B 0,C 180,E1 35304.792,E2 35304.792} C_VEL
LIN {X 0,Y 19.335,Z 1169.516,A -85,B 0,C 180,E1 35421.439,E2 35421.439} C_VEL
LIN {X 0,Y 46.965,Z 1165.641,A -85,B 0,C 180,E1 35444.89,E2 35444.89} C_VEL
LIN {X 0,Y 61.473,Z 1163.008,A -85,B 0,C 180,E1 35449.544,E2 35449.544} C_VEL
LIN {X 0,Y 70.821,Z 1161.259,A -85,B 0,C 180,E1 35452.743,E2 35452.743} C_VEL
LIN {X 0,Y 36.79,Z 1168.319,A -85,B 0,C 180,E1 35463.088,E2 35463.088} C_VEL
LIN {X 0,Y 23.877,Z 1169.972,A -85,B 0,C 180,E1 35466.63,E2 35466.63} C_VEL
LIN {X 0,Y 2.383,Z 1171.671,A -85,B 0,C 180,E1 35506.396,E2 35506.396} C_VEL
LIN {X 0,Y 9.84,Z 1172.038,A -85,B 0,C 180,E1 35640.243,E2 35640.243} C_VEL
LIN {X 0,Y 15.668,Z 1170.244,A -85,B 0,C 180,E1 35804.789,E2 35804.789} C_VEL
LIN {X 0,Y 30.546,Z 1168.592,A -85,B 0,C 180,E1 35811.754,E2 35811.754} C_VEL
LIN {X 0,Y 2.383,Z 1171.671,A -85,B 0,C 180,E1 35866.396,E2 35866.396} C_VEL
LIN {X 0,Y 2.045,Z 1173.665,A -85,B 0,C 180,E1 35914.998,E2 35914.998} C_VEL
LIN {X 0,Y 2.045,Z 1215,A -85,B 0,C 180,E1 35914.998,E2 35914.998} C_VEL
LIN {X 0,Y 2.045,Z 1215,A -85,B 0,C 180,E1 35914.998,E2 35914.998}

